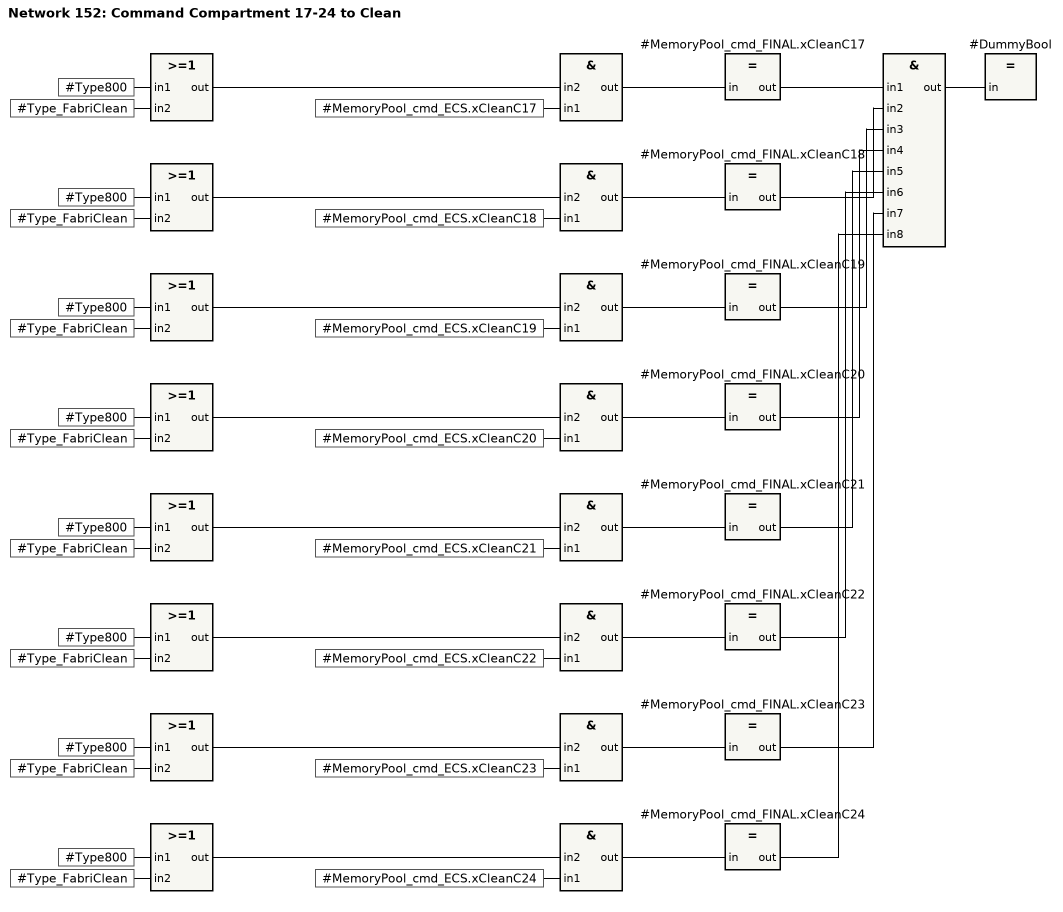
   #MemoryPool_cmd_FINAL.xCleanC17 := (#Type800 OR #Type_FabriClean) AND #MemoryPool_cmd_ECS.xCleanC17;
   #MemoryPool_cmd_FINAL.xCleanC18 := (#Type800 OR #Type_FabriClean) AND #MemoryPool_cmd_ECS.xCleanC18;
   #MemoryPool_cmd_FINAL.xCleanC19 := (#Type800 OR #Type_FabriClean) AND #MemoryPool_cmd_ECS.xCleanC19;
   #MemoryPool_cmd_FINAL.xCleanC20 := (#Type800 OR #Type_FabriClean) AND #MemoryPool_cmd_ECS.xCleanC20;
   #MemoryPool_cmd_FINAL.xCleanC21 := (#Type800 OR #Type_FabriClean) AND #MemoryPool_cmd_ECS.xCleanC21;
   #MemoryPool_cmd_FINAL.xCleanC22 := (#Type800 OR #Type_FabriClean) AND #MemoryPool_cmd_ECS.xCleanC22;
   #MemoryPool_cmd_FINAL.xCleanC23 := (#Type800 OR #Type_FabriClean) AND #MemoryPool_cmd_ECS.xCleanC23;
   #MemoryPool_cmd_FINAL.xCleanC24 := (#Type800 OR #Type_FabriClean) AND #MemoryPool_cmd_ECS.xCleanC24;
   #DummyBool := #MemoryPool_cmd_FINAL.xCleanC17 AND #MemoryPool_cmd_FINAL.xCleanC18 AND #MemoryPool_cmd_FINAL.xCleanC19 AND #MemoryPool_cmd_FINAL.xCleanC20 AND #MemoryPool_cmd_FINAL.xCleanC21 AND #MemoryPool_cmd_FINAL.xCleanC22 AND #MemoryPool_cmd_FINAL.xCleanC23 AND #MemoryPool_cmd_FINAL.xCleanC24;
END_REGION

REGION Network 153: Reset Clean Command 1-8
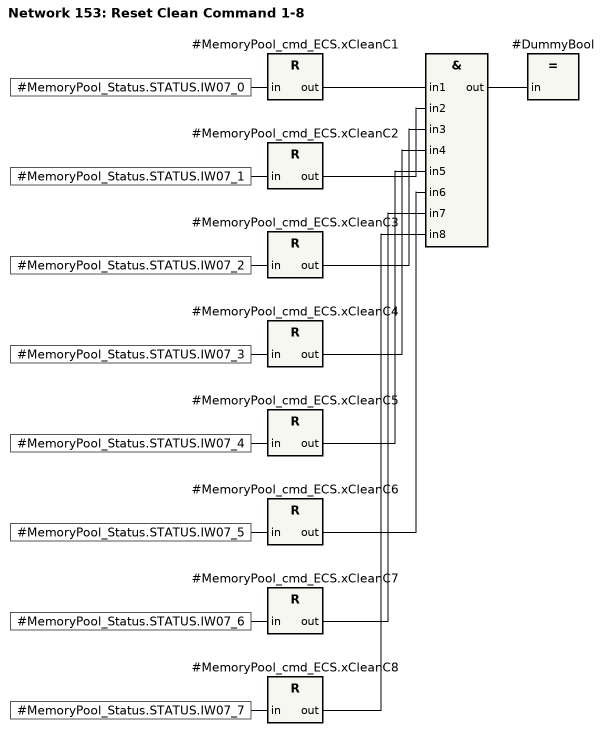
   IF #MemoryPool_Status.STATUS.IW07_0 THEN #MemoryPool_cmd_ECS.xCleanC1 := FALSE; END_IF;
   IF #MemoryPool_Status.STATUS.IW07_1 THEN #MemoryPool_cmd_ECS.xCleanC2 := FALSE; END_IF;
   IF #MemoryPool_Status.STATUS.IW07_2 THEN #MemoryPool_cmd_ECS.xCleanC3 := FALSE; END_IF;
   IF #MemoryPool_Status.STATUS.IW07_3 THEN #MemoryPool_cmd_ECS.xCleanC4 := FALSE; END_IF;
   IF #MemoryPool_Status.STATUS.IW07_4 THEN #MemoryPool_cmd_ECS.xCleanC5 := FALSE; END_IF;
   IF #MemoryPool_Status.STATUS.IW07_5 THEN #MemoryPool_cmd_ECS.xCleanC6 := FALSE; END_IF;
   IF #MemoryPool_Status.STATUS.IW07_6 THEN #MemoryPool_cmd_ECS.xCleanC7 := FALSE; END_IF;
   IF #MemoryPool_Status.STATUS.IW07_7 THEN #MemoryPool_cmd_ECS.xCleanC8 := FALSE; END_IF;
   #DummyBool := #MemoryPool_Status.STATUS.IW07_0 AND #MemoryPool_Status.STATUS.IW07_1 AND #MemoryPool_Status.STATUS.IW07_2 AND #MemoryPool_Status.STATUS.IW07_3 AND #MemoryPool_Status.STATUS.IW07_4 AND #MemoryPool_Status.STATUS.IW07_5 AND #MemoryPool_Status.STATUS.IW07_6 AND #MemoryPool_Status.STATUS.IW07_7;
END_REGION

REGION Network 154: Reset Clean Command 9-16
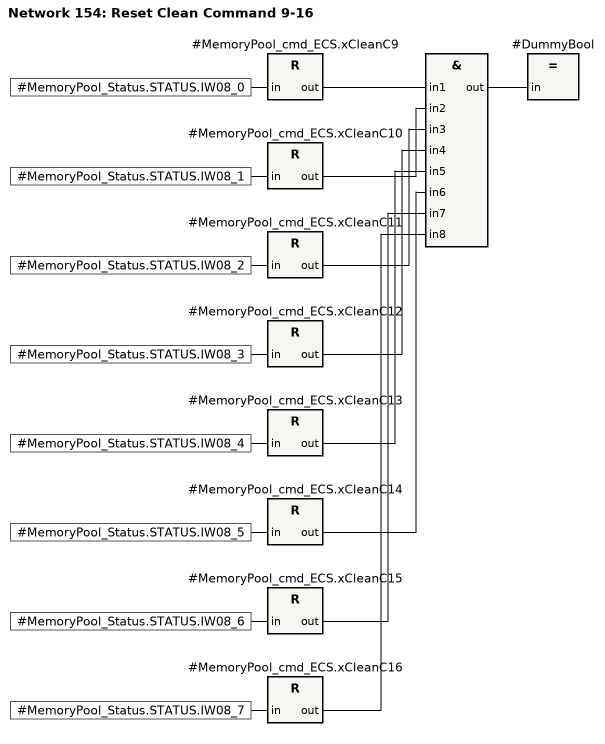
   IF #MemoryPool_Status.STATUS.IW08_0 THEN #MemoryPool_cmd_ECS.xCleanC9 := FALSE; END_IF;
   IF #MemoryPool_Status.STATUS.IW08_1 THEN #MemoryPool_cmd_ECS.xCleanC10 := FALSE; END_IF;
   IF #MemoryPool_Status.STATUS.IW08_2 THEN #MemoryPool_cmd_ECS.xCleanC11 := FALSE; END_IF;
   IF #MemoryPool_Status.STATUS.IW08_3 THEN #MemoryPool_cmd_ECS.xCleanC12 := FALSE; END_IF;
   IF #MemoryPool_Status.STATUS.IW08_4 THEN #MemoryPool_cmd_ECS.xCleanC13 := FALSE; END_IF;
   IF #MemoryPool_Status.STATUS.IW08_5 THEN #MemoryPool_cmd_ECS.xCleanC14 := FALSE; END_IF;
   IF #MemoryPool_Status.STATUS.IW08_6 THEN #MemoryPool_cmd_ECS.xCleanC15 := FALSE; END_IF;
   IF #MemoryPool_Status.STATUS.IW08_7 THEN #MemoryPool_cmd_ECS.xCleanC16 := FALSE; END_IF;
   #DummyBool := #MemoryPool_Status.STATUS.IW08_0 AND #MemoryPool_Status.STATUS.IW08_1 AND #MemoryPool_Status.STATUS.IW08_2 AND #MemoryPool_Status.STATUS.IW08_3 AND #MemoryPool_Status.STATUS.IW08_4 AND #MemoryPool_Status.STATUS.IW08_5 AND #MemoryPool_Status.STATUS.IW08_6 AND #MemoryPool_Status.STATUS.IW08_7;
END_REGION

REGION Network 155: Reset Clean Command 17-24
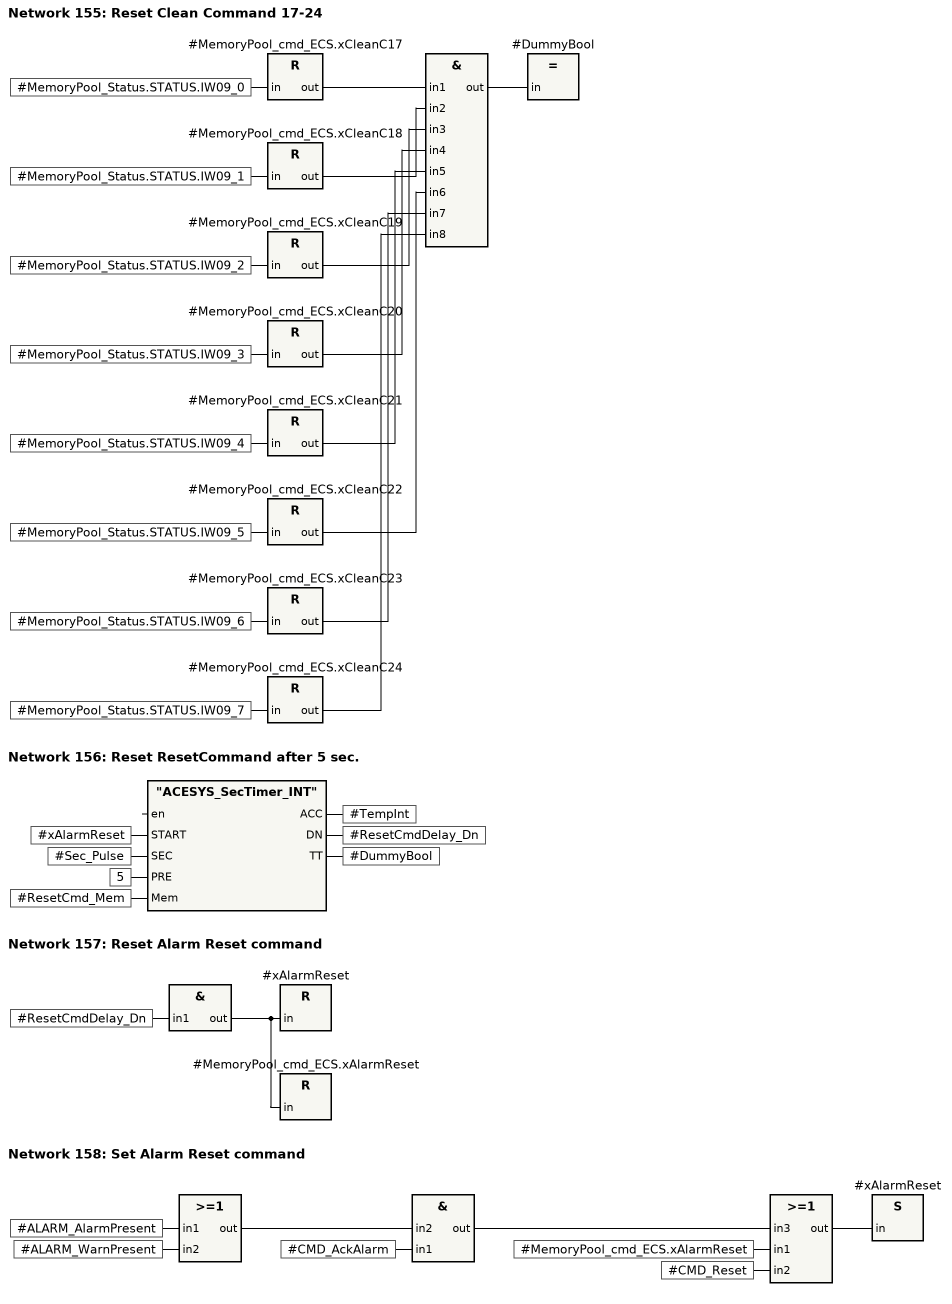
   IF #MemoryPool_Status.STATUS.IW09_0 THEN #MemoryPool_cmd_ECS.xCleanC17 := FALSE; END_IF;
   IF #MemoryPool_Status.STATUS.IW09_1 THEN #MemoryPool_cmd_ECS.xCleanC18 := FALSE; END_IF;
   IF #MemoryPool_Status.STATUS.IW09_2 THEN #MemoryPool_cmd_ECS.xCleanC19 := FALSE; END_IF;
   IF #MemoryPool_Status.STATUS.IW09_3 THEN #MemoryPool_cmd_ECS.xCleanC20 := FALSE; END_IF;
   IF #MemoryPool_Status.STATUS.IW09_4 THEN #MemoryPool_cmd_ECS.xCleanC21 := FALSE; END_IF;
   IF #MemoryPool_Status.STATUS.IW09_5 THEN #MemoryPool_cmd_ECS.xCleanC22 := FALSE; END_IF;
   IF #MemoryPool_Status.STATUS.IW09_6 THEN #MemoryPool_cmd_ECS.xCleanC23 := FALSE; END_IF;
   IF #MemoryPool_Status.STATUS.IW09_7 THEN #MemoryPool_cmd_ECS.xCleanC24 := FALSE; END_IF;
   #DummyBool := #MemoryPool_Status.STATUS.IW09_0 AND #MemoryPool_Status.STATUS.IW09_1 AND #MemoryPool_Status.STATUS.IW09_2 AND #MemoryPool_Status.STATUS.IW09_3 AND #MemoryPool_Status.STATUS.IW09_4 AND #MemoryPool_Status.STATUS.IW09_5 AND #MemoryPool_Status.STATUS.IW09_6 AND #MemoryPool_Status.STATUS.IW09_7;
END_REGION

REGION Network 156: Reset ResetCommand after 5 sec.
   "ACESYS_SecTimer_INT"(START := #xAlarmReset,
                         SEC := #Sec_Pulse,
                         PRE := 5,
                         Mem := #ResetCmd_Mem,
                         ACC => #TempInt,
                         DN => #ResetCmdDelay_Dn,
                         TT => #DummyBool);
END_REGION

REGION Network 157: Reset Alarm Reset command
   IF #ResetCmdDelay_Dn THEN
       #xAlarmReset := FALSE;
       #MemoryPool_cmd_ECS.xAlarmReset := FALSE;
   END_IF;
END_REGION

REGION Network 158: Set Alarm Reset command
   IF ((#ALARM_AlarmPresent OR #ALARM_WarnPresent) AND #CMD_AckAlarm) OR #MemoryPool_cmd_ECS.xAlarmReset OR #CMD_Reset THEN
       #xAlarmReset := TRUE;
   END_IF;
END_REGION

REGION Network 159
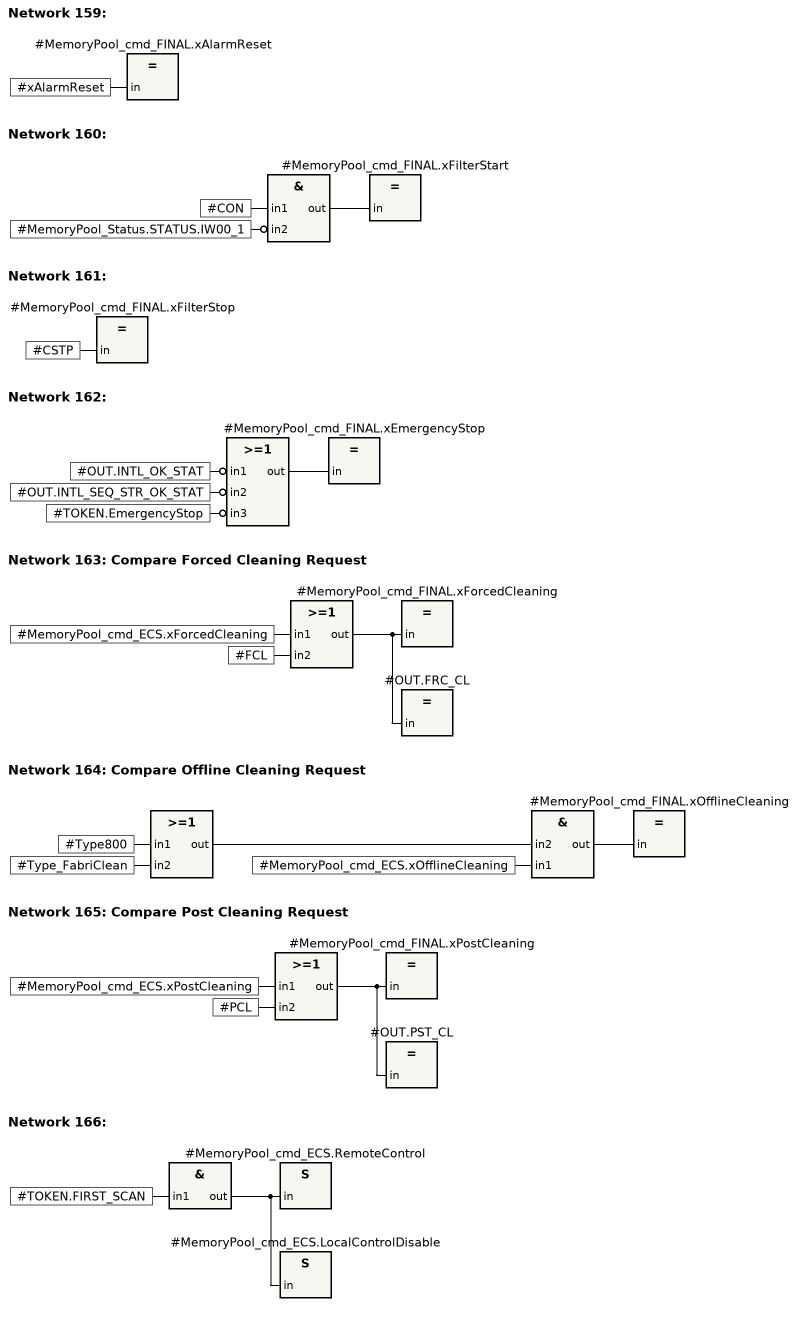
   #MemoryPool_cmd_FINAL.xAlarmReset := #xAlarmReset;
END_REGION

REGION Network 160
   #MemoryPool_cmd_FINAL.xFilterStart := #CON AND NOT #MemoryPool_Status.STATUS.IW00_1;
END_REGION

REGION Network 161
   #MemoryPool_cmd_FINAL.xFilterStop := #CSTP;
END_REGION

REGION Network 162
   #MemoryPool_cmd_FINAL.xEmergencyStop := NOT #OUT.INTL_OK_STAT OR NOT #OUT.INTL_SEQ_STR_OK_STAT OR NOT #TOKEN.EmergencyStop;
END_REGION

REGION Network 163: Compare Forced Cleaning Request
   #MemoryPool_cmd_FINAL.xForcedCleaning := #MemoryPool_cmd_ECS.xForcedCleaning OR #FCL;
   #OUT.FRC_CL := #MemoryPool_cmd_FINAL.xForcedCleaning;
END_REGION

REGION Network 164: Compare Offline Cleaning Request
   #MemoryPool_cmd_FINAL.xOfflineCleaning := (#Type800 OR #Type_FabriClean) AND #MemoryPool_cmd_ECS.xOfflineCleaning;
END_REGION

REGION Network 165: Compare Post Cleaning Request
   #MemoryPool_cmd_FINAL.xPostCleaning := #MemoryPool_cmd_ECS.xPostCleaning OR #PCL;
   #OUT.PST_CL := #MemoryPool_cmd_FINAL.xPostCleaning;
END_REGION

REGION Network 166
   IF #TOKEN.FIRST_SCAN THEN
       #MemoryPool_cmd_ECS.RemoteControl := TRUE;
       #MemoryPool_cmd_ECS.LocalControlDisable := TRUE;
   END_IF;
END_REGION

REGION Network 167
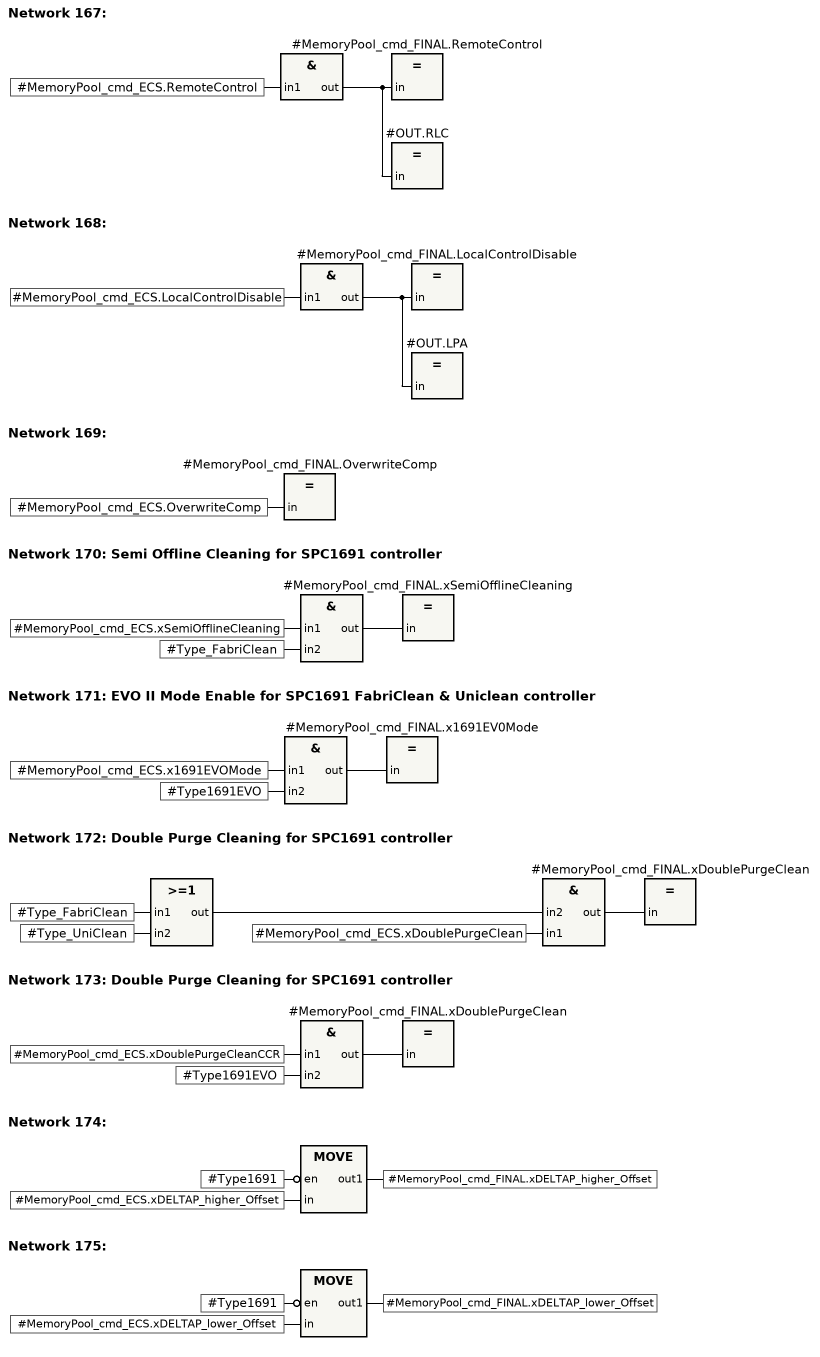
   #MemoryPool_cmd_FINAL.RemoteControl := #MemoryPool_cmd_ECS.RemoteControl;
   #OUT.RLC := #MemoryPool_cmd_ECS.RemoteControl;
END_REGION

REGION Network 168
   #MemoryPool_cmd_FINAL.LocalControlDisable := #MemoryPool_cmd_ECS.LocalControlDisable;
   #OUT.LPA := #MemoryPool_cmd_ECS.LocalControlDisable;
END_REGION

REGION Network 169
   #MemoryPool_cmd_FINAL.OverwriteComp := #MemoryPool_cmd_ECS.OverwriteComp;
END_REGION

REGION Network 170: Semi Offline Cleaning for SPC1691 controller
   #MemoryPool_cmd_FINAL.xSemiOfflineCleaning := #MemoryPool_cmd_ECS.xSemiOfflineCleaning AND #Type_FabriClean;
END_REGION

REGION Network 171: EVO II Mode Enable for SPC1691 FabriClean & Uniclean controller
   // Build 007 - 03.12.2020 (VIV-IN): EVO II Mode Enable for SPC1691 FabriClean & 
   // UniClean controller - Newly Added
   #MemoryPool_cmd_FINAL.x1691EV0Mode := #MemoryPool_cmd_ECS.x1691EVOMode AND #Type1691EVO;
END_REGION

REGION Network 172: Double Purge Cleaning for SPC1691 controller
   // Build 007 - 03.12.2020 (VIV-IN): Type UniClean also added
   #MemoryPool_cmd_FINAL.xDoublePurgeClean := (#Type_FabriClean OR #Type_UniClean) AND #MemoryPool_cmd_ECS.xDoublePurgeClean;
END_REGION

REGION Network 173: Double Purge Cleaning for SPC1691 controller
   // Build 007 - 03.12.2020 (VIV-IN): EVO Mode Double Purge Cleaning Continuous 
   // Cycle Request for SPC1691 FabriClean and UniClean controller - Newly Added
   #MemoryPool_cmd_FINAL.xDoublePurgeClean := #MemoryPool_cmd_ECS.xDoublePurgeCleanCCR AND #Type1691EVO;
END_REGION

REGION Network 174
   IF NOT #Type1691 THEN
       #MemoryPool_cmd_FINAL.xDELTAP_higher_Offset := #MemoryPool_cmd_ECS.xDELTAP_higher_Offset;
   END_IF;
END_REGION

REGION Network 175
   IF NOT #Type1691 THEN
       #MemoryPool_cmd_FINAL.xDELTAP_lower_Offset := #MemoryPool_cmd_ECS.xDELTAP_lower_Offset;
   END_IF;
END_REGION

REGION Network 176
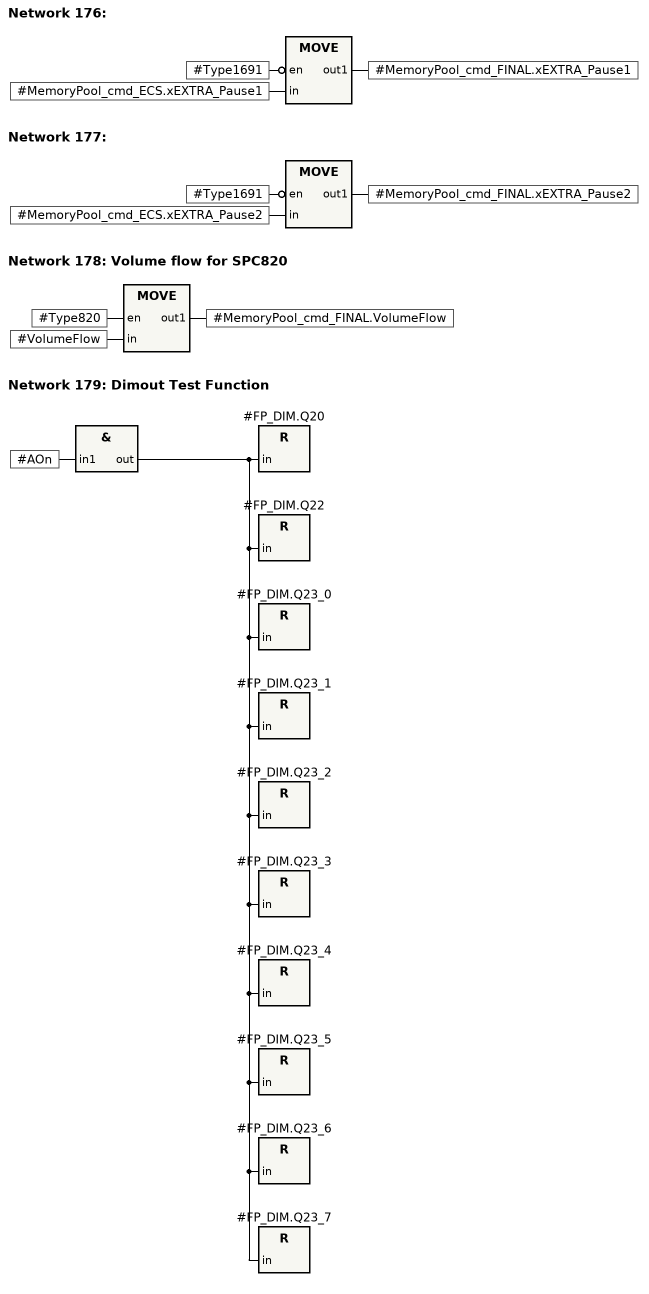
   IF NOT #Type1691 THEN #MemoryPool_cmd_FINAL.xEXTRA_Pause1 := #MemoryPool_cmd_ECS.xEXTRA_Pause1; END_IF;
END_REGION

REGION Network 177
   IF NOT #Type1691 THEN #MemoryPool_cmd_FINAL.xEXTRA_Pause2 := #MemoryPool_cmd_ECS.xEXTRA_Pause2; END_IF;
END_REGION

REGION Network 178: Volume flow for SPC820
   IF #Type820 THEN #MemoryPool_cmd_FINAL.VolumeFlow := #VolumeFlow; END_IF;
END_REGION

REGION Network 179: Dimout Test Function
   IF #AOn THEN
       #FP_DIM.Q20 := FALSE;
       #FP_DIM.Q22 := FALSE;
       #FP_DIM.Q23_0 := FALSE;
       #FP_DIM.Q23_1 := FALSE;
       #FP_DIM.Q23_2 := FALSE;
       #FP_DIM.Q23_3 := FALSE;
       #FP_DIM.Q23_4 := FALSE;
       #FP_DIM.Q23_5 := FALSE;
       #FP_DIM.Q23_6 := FALSE;
       #FP_DIM.Q23_7 := FALSE;
   END_IF;
END_REGION

REGION Network 180: Dimout test values/commands
   // Check for compartment number typed in
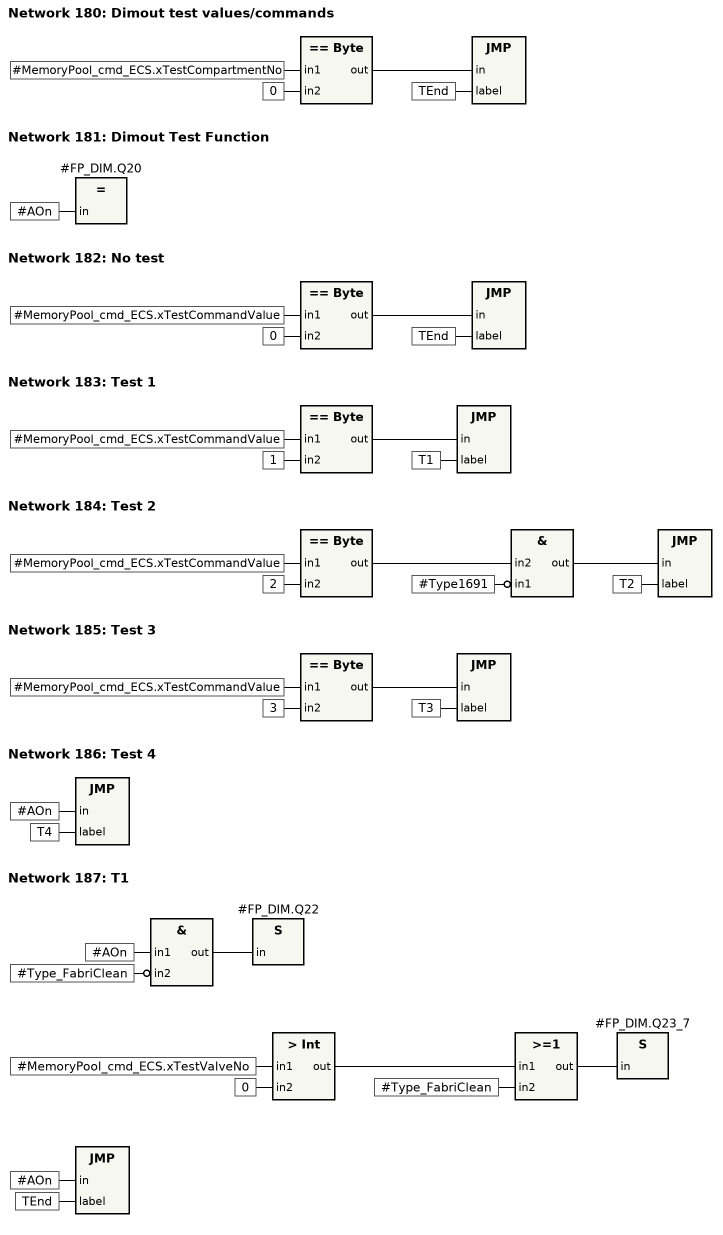
   IF #MemoryPool_cmd_ECS.xTestCompartmentNo = 0 THEN GOTO TEnd; END_IF;
END_REGION

REGION Network 181: Dimout Test Function
   #FP_DIM.Q20 := #AOn;
END_REGION

REGION Network 182: No test
   IF #MemoryPool_cmd_ECS.xTestCommandValue = 0 THEN GOTO TEnd; END_IF;
END_REGION

REGION Network 183: Test 1
   IF #MemoryPool_cmd_ECS.xTestCommandValue = 1 THEN GOTO T1; END_IF;
END_REGION

REGION Network 184: Test 2
   IF (#MemoryPool_cmd_ECS.xTestCommandValue = 2) AND NOT #Type1691 THEN GOTO T2; END_IF;
END_REGION

REGION Network 185: Test 3
   IF #MemoryPool_cmd_ECS.xTestCommandValue = 3 THEN GOTO T3; END_IF;
END_REGION

REGION Network 186: Test 4
   IF #AOn THEN GOTO T4; END_IF;
END_REGION

REGION Network 187: T1
   T1:
   IF #AOn AND NOT #Type_FabriClean THEN #FP_DIM.Q22 := TRUE; END_IF;
   IF (#MemoryPool_cmd_ECS.xTestValveNo > 0) OR #Type_FabriClean THEN #FP_DIM.Q23_7 := TRUE; END_IF;
   IF #AOn THEN GOTO TEnd; END_IF;
END_REGION

REGION Network 188: T2
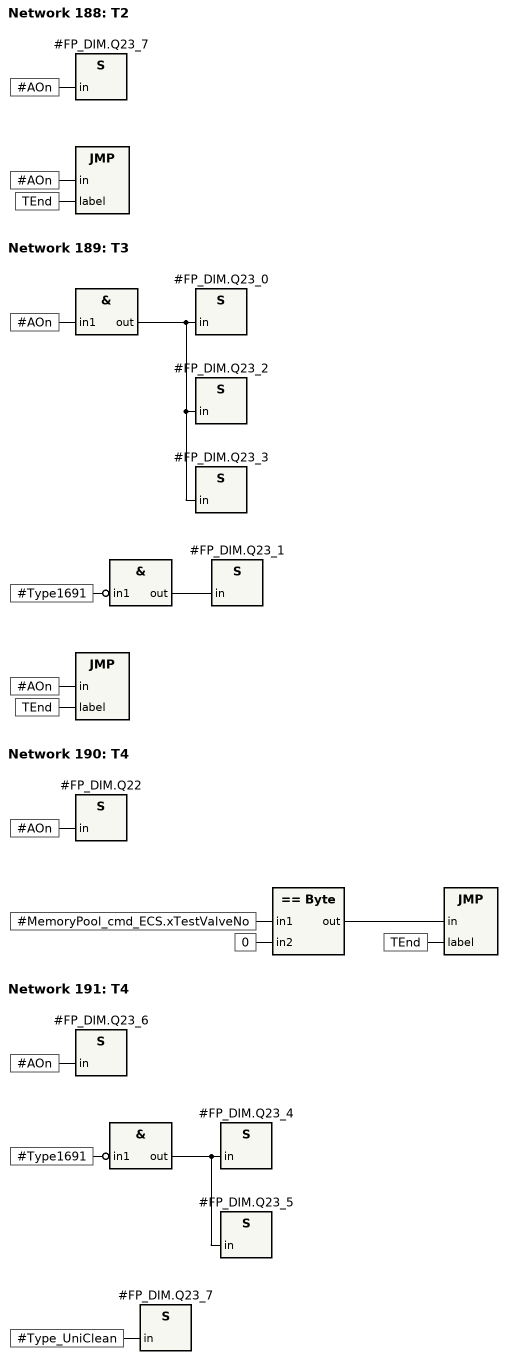
   T2:
   IF #AOn THEN
       #FP_DIM.Q23_7 := TRUE;
       GOTO TEnd;
   END_IF;
END_REGION

REGION Network 189: T3
   T3:
   IF #AOn THEN
       #FP_DIM.Q23_0 := TRUE;
       #FP_DIM.Q23_2 := TRUE;
       #FP_DIM.Q23_3 := TRUE;
   END_IF;
   IF NOT #Type1691 THEN #FP_DIM.Q23_1 := TRUE; END_IF;
   IF #AOn THEN GOTO TEnd; END_IF;
END_REGION

REGION Network 190: T4
   T4:
   IF #AOn THEN #FP_DIM.Q22 := TRUE; END_IF;
   IF #MemoryPool_cmd_ECS.xTestValveNo = 0 THEN GOTO TEnd; END_IF;
END_REGION

REGION Network 191: T4
   IF #AOn THEN #FP_DIM.Q23_6 := TRUE; END_IF;
   IF NOT #Type1691 THEN
       #FP_DIM.Q23_4 := TRUE;
       #FP_DIM.Q23_5 := TRUE;
   END_IF;
   IF #Type_UniClean THEN #FP_DIM.Q23_7 := TRUE; END_IF;
END_REGION

REGION Network 192
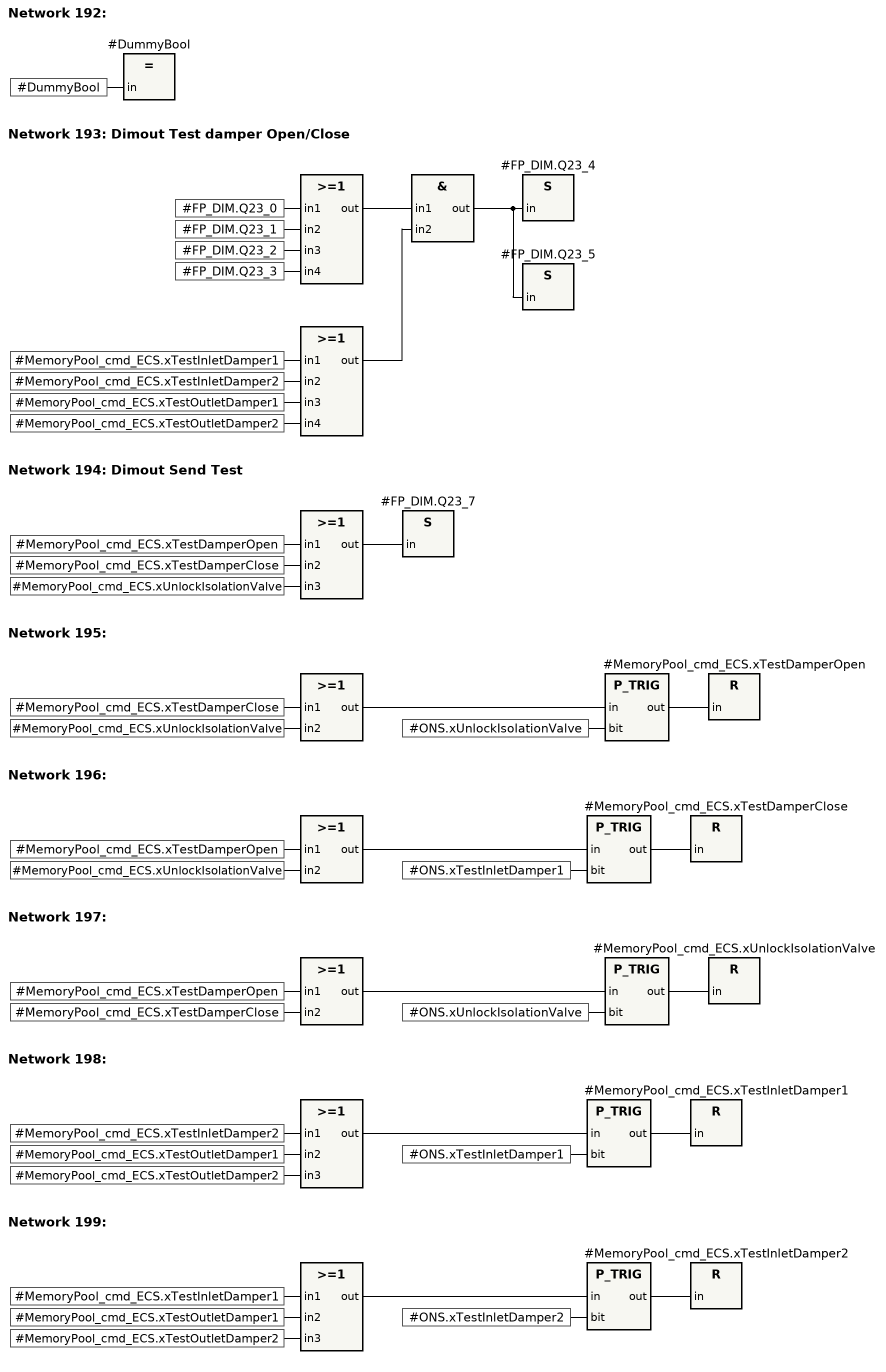
   TEnd:
   #DummyBool := #DummyBool;
END_REGION

REGION Network 193: Dimout Test damper Open/Close
   IF (#FP_DIM.Q23_0 OR #FP_DIM.Q23_1 OR #FP_DIM.Q23_2 OR #FP_DIM.Q23_3) AND (#MemoryPool_cmd_ECS.xTestInletDamper1 OR #MemoryPool_cmd_ECS.xTestInletDamper2 OR #MemoryPool_cmd_ECS.xTestOutletDamper1 OR #MemoryPool_cmd_ECS.xTestOutletDamper2) THEN
       #FP_DIM.Q23_4 := TRUE;
       #FP_DIM.Q23_5 := TRUE;
   END_IF;
END_REGION

REGION Network 194: Dimout Send Test
   IF #MemoryPool_cmd_ECS.xTestDamperOpen OR #MemoryPool_cmd_ECS.xTestDamperClose OR #MemoryPool_cmd_ECS.xUnlockIsolationValve THEN
       #FP_DIM.Q23_7 := TRUE;
   END_IF;
END_REGION

REGION Network 195
   #_w1 := #MemoryPool_cmd_ECS.xTestDamperClose OR #MemoryPool_cmd_ECS.xUnlockIsolationValve;
   #_w2 := #_w1 AND NOT #ONS.xUnlockIsolationValve;   // rising edge
   #ONS.xUnlockIsolationValve := #_w1;
   IF #_w2 THEN #MemoryPool_cmd_ECS.xTestDamperOpen := FALSE; END_IF;
END_REGION

REGION Network 196
   #_w1 := #MemoryPool_cmd_ECS.xTestDamperOpen OR #MemoryPool_cmd_ECS.xUnlockIsolationValve;
   #_w2 := #_w1 AND NOT #ONS.xTestInletDamper1;   // rising edge
   #ONS.xTestInletDamper1 := #_w1;
   IF #_w2 THEN #MemoryPool_cmd_ECS.xTestDamperClose := FALSE; END_IF;
END_REGION

REGION Network 197
   #_w1 := #MemoryPool_cmd_ECS.xTestDamperOpen OR #MemoryPool_cmd_ECS.xTestDamperClose;
   #_w2 := #_w1 AND NOT #ONS.xUnlockIsolationValve;   // rising edge
   #ONS.xUnlockIsolationValve := #_w1;
   IF #_w2 THEN #MemoryPool_cmd_ECS.xUnlockIsolationValve := FALSE; END_IF;
END_REGION

REGION Network 198
   #_w1 := #MemoryPool_cmd_ECS.xTestInletDamper2 OR #MemoryPool_cmd_ECS.xTestOutletDamper1 OR #MemoryPool_cmd_ECS.xTestOutletDamper2;
   #_w2 := #_w1 AND NOT #ONS.xTestInletDamper1;   // rising edge
   #ONS.xTestInletDamper1 := #_w1;
   IF #_w2 THEN #MemoryPool_cmd_ECS.xTestInletDamper1 := FALSE; END_IF;
END_REGION

REGION Network 199
   #_w1 := #MemoryPool_cmd_ECS.xTestInletDamper1 OR #MemoryPool_cmd_ECS.xTestOutletDamper1 OR #MemoryPool_cmd_ECS.xTestOutletDamper2;
   #_w2 := #_w1 AND NOT #ONS.xTestInletDamper2;   // rising edge
   #ONS.xTestInletDamper2 := #_w1;
   IF #_w2 THEN #MemoryPool_cmd_ECS.xTestInletDamper2 := FALSE; END_IF;
END_REGION

REGION Network 200
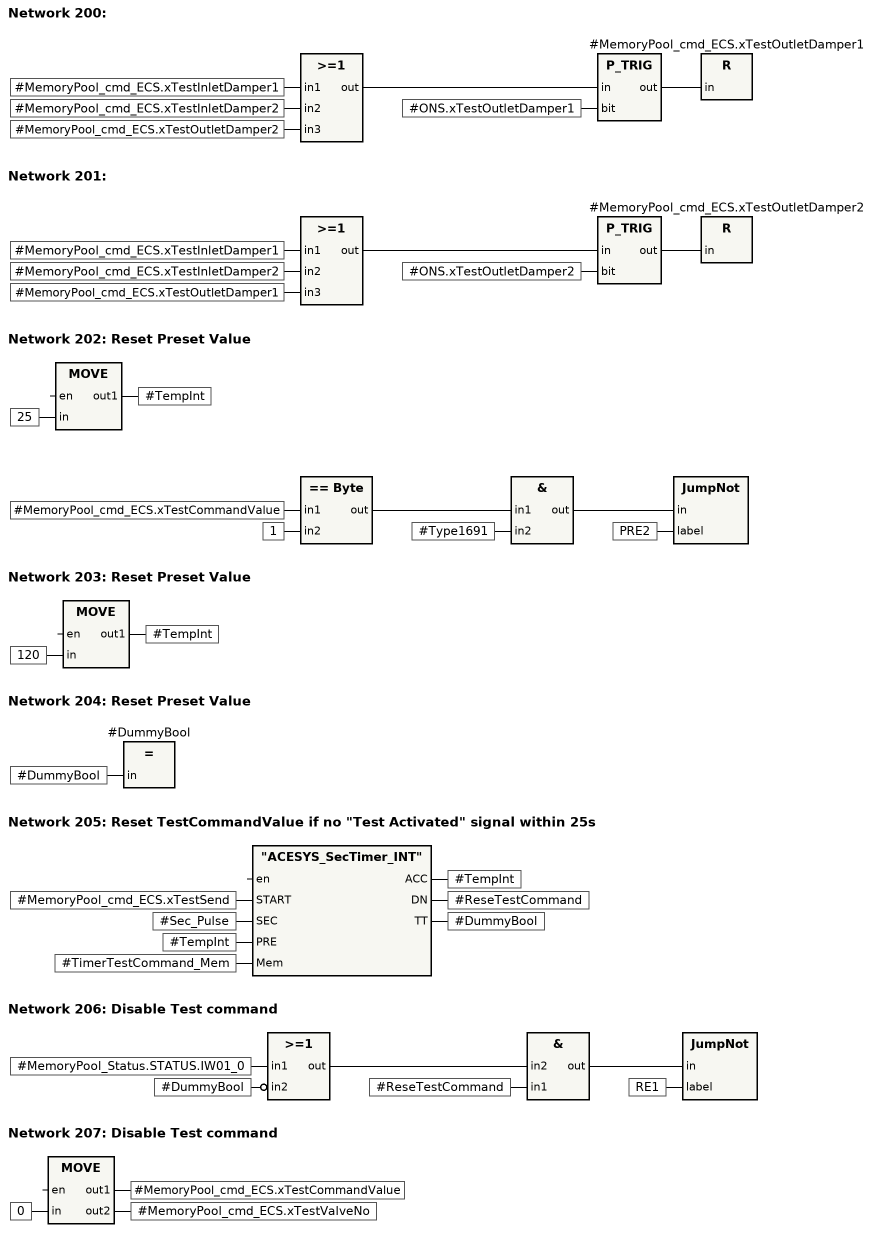
   #_w1 := #MemoryPool_cmd_ECS.xTestInletDamper1 OR #MemoryPool_cmd_ECS.xTestInletDamper2 OR #MemoryPool_cmd_ECS.xTestOutletDamper2;
   #_w2 := #_w1 AND NOT #ONS.xTestOutletDamper1;   // rising edge
   #ONS.xTestOutletDamper1 := #_w1;
   IF #_w2 THEN #MemoryPool_cmd_ECS.xTestOutletDamper1 := FALSE; END_IF;
END_REGION

REGION Network 201
   #_w1 := #MemoryPool_cmd_ECS.xTestInletDamper1 OR #MemoryPool_cmd_ECS.xTestInletDamper2 OR #MemoryPool_cmd_ECS.xTestOutletDamper1;
   #_w2 := #_w1 AND NOT #ONS.xTestOutletDamper2;   // rising edge
   #ONS.xTestOutletDamper2 := #_w1;
   IF #_w2 THEN #MemoryPool_cmd_ECS.xTestOutletDamper2 := FALSE; END_IF;
END_REGION

REGION Network 202: Reset Preset Value
   // - SPC1691 =>120s
   // - Hesch   =>25s
   // no SCL statement known for JumpNot: written as a call
   #TempInt := 25;
   JumpNot(in := (#MemoryPool_cmd_ECS.xTestCommandValue = 1) AND #Type1691, label := PRE2);
END_REGION

REGION Network 203: Reset Preset Value
   #TempInt := 120;
END_REGION

REGION Network 204: Reset Preset Value
   PRE2:
   #DummyBool := #DummyBool;
END_REGION

REGION Network 205: Reset TestCommandValue if no "Test Activated" signal within 25s
   "ACESYS_SecTimer_INT"(START := #MemoryPool_cmd_ECS.xTestSend,
                         SEC := #Sec_Pulse,
                         PRE := #TempInt,
                         Mem := #TimerTestCommand_Mem,
                         ACC => #TempInt,
                         DN => #ReseTestCommand,
                         TT => #DummyBool);
END_REGION

REGION Network 206: Disable Test command
   // Disable Test command once test activated is completed. This 
   // ensures that the command value is not always sent to the SPC
   // no SCL statement known for JumpNot: written as a call
   JumpNot(in := (#MemoryPool_Status.STATUS.IW01_0 OR NOT #DummyBool) AND #ReseTestCommand, label := RE1);
END_REGION

REGION Network 207: Disable Test command
   #MemoryPool_cmd_ECS.xTestCommandValue := 0;
   #MemoryPool_cmd_ECS.xTestValveNo := 0;
END_REGION

REGION Network 208: Disable Test command
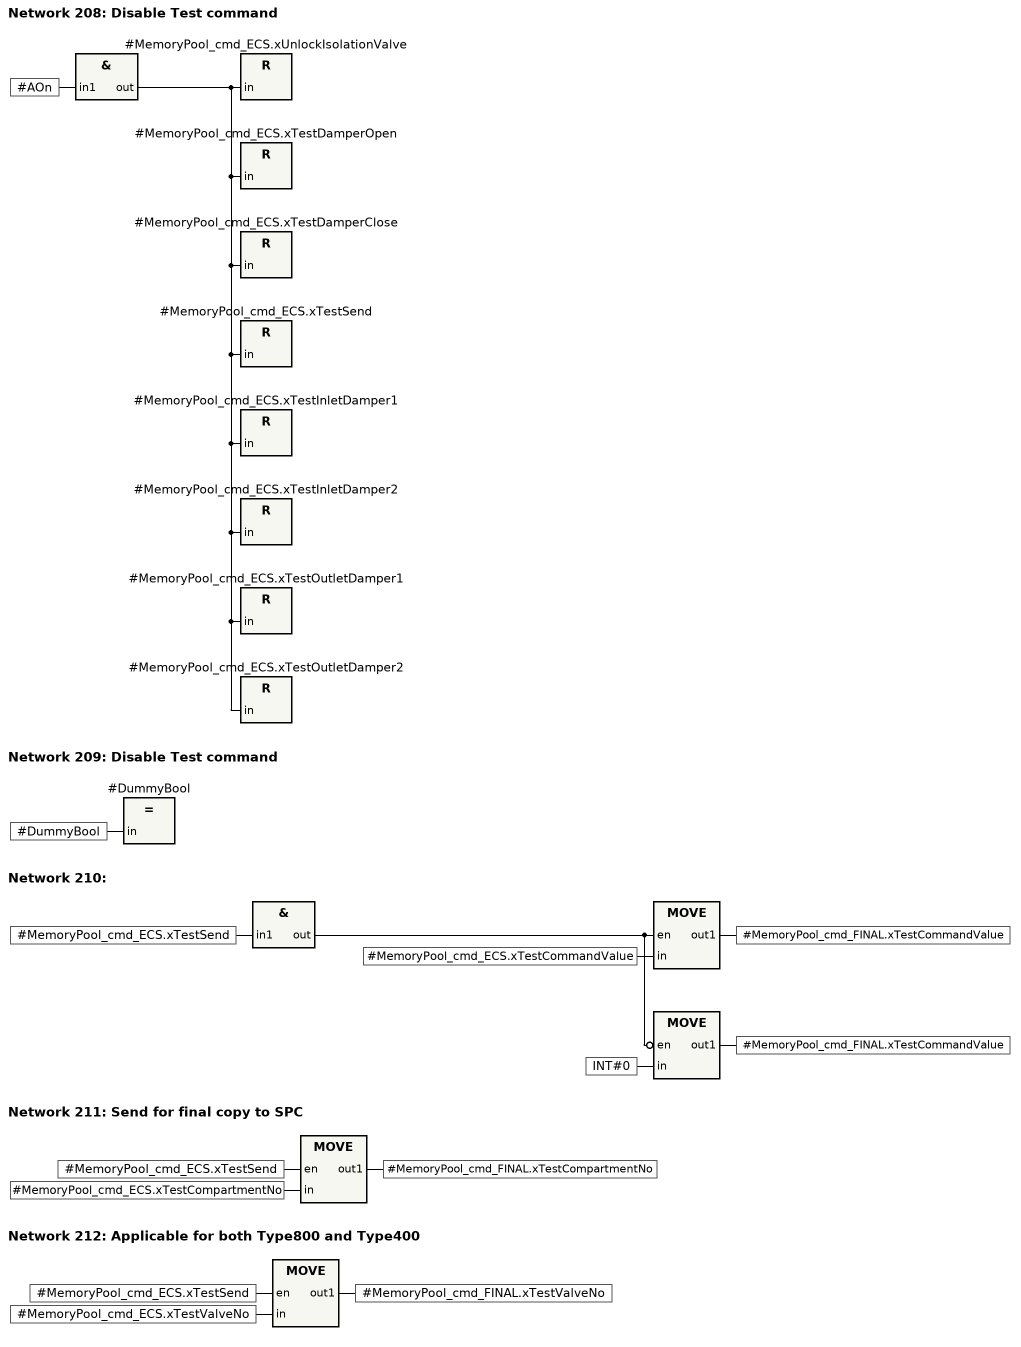
   IF #AOn THEN
       #MemoryPool_cmd_ECS.xUnlockIsolationValve := FALSE;
       #MemoryPool_cmd_ECS.xTestDamperOpen := FALSE;
       #MemoryPool_cmd_ECS.xTestDamperClose := FALSE;
       #MemoryPool_cmd_ECS.xTestSend := FALSE;
       #MemoryPool_cmd_ECS.xTestInletDamper1 := FALSE;
       #MemoryPool_cmd_ECS.xTestInletDamper2 := FALSE;
       #MemoryPool_cmd_ECS.xTestOutletDamper1 := FALSE;
       #MemoryPool_cmd_ECS.xTestOutletDamper2 := FALSE;
   END_IF;
END_REGION

REGION Network 209: Disable Test command
   RE1:
   #DummyBool := #DummyBool;
END_REGION

REGION Network 210
   IF #MemoryPool_cmd_ECS.xTestSend THEN
       #MemoryPool_cmd_FINAL.xTestCommandValue := #MemoryPool_cmd_ECS.xTestCommandValue;
   END_IF;
   IF NOT #MemoryPool_cmd_ECS.xTestSend THEN #MemoryPool_cmd_FINAL.xTestCommandValue := INT#0; END_IF;
END_REGION

REGION Network 211: Send for final copy to SPC
   // Applicable for Type 800 and 400. Type 400 is refered to as section
   IF #MemoryPool_cmd_ECS.xTestSend THEN
       #MemoryPool_cmd_FINAL.xTestCompartmentNo := #MemoryPool_cmd_ECS.xTestCompartmentNo;
   END_IF;
END_REGION

REGION Network 212: Applicable for both Type800 and Type400
   IF #MemoryPool_cmd_ECS.xTestSend THEN
       #MemoryPool_cmd_FINAL.xTestValveNo := #MemoryPool_cmd_ECS.xTestValveNo;
   END_IF;
END_REGION

REGION Network 213
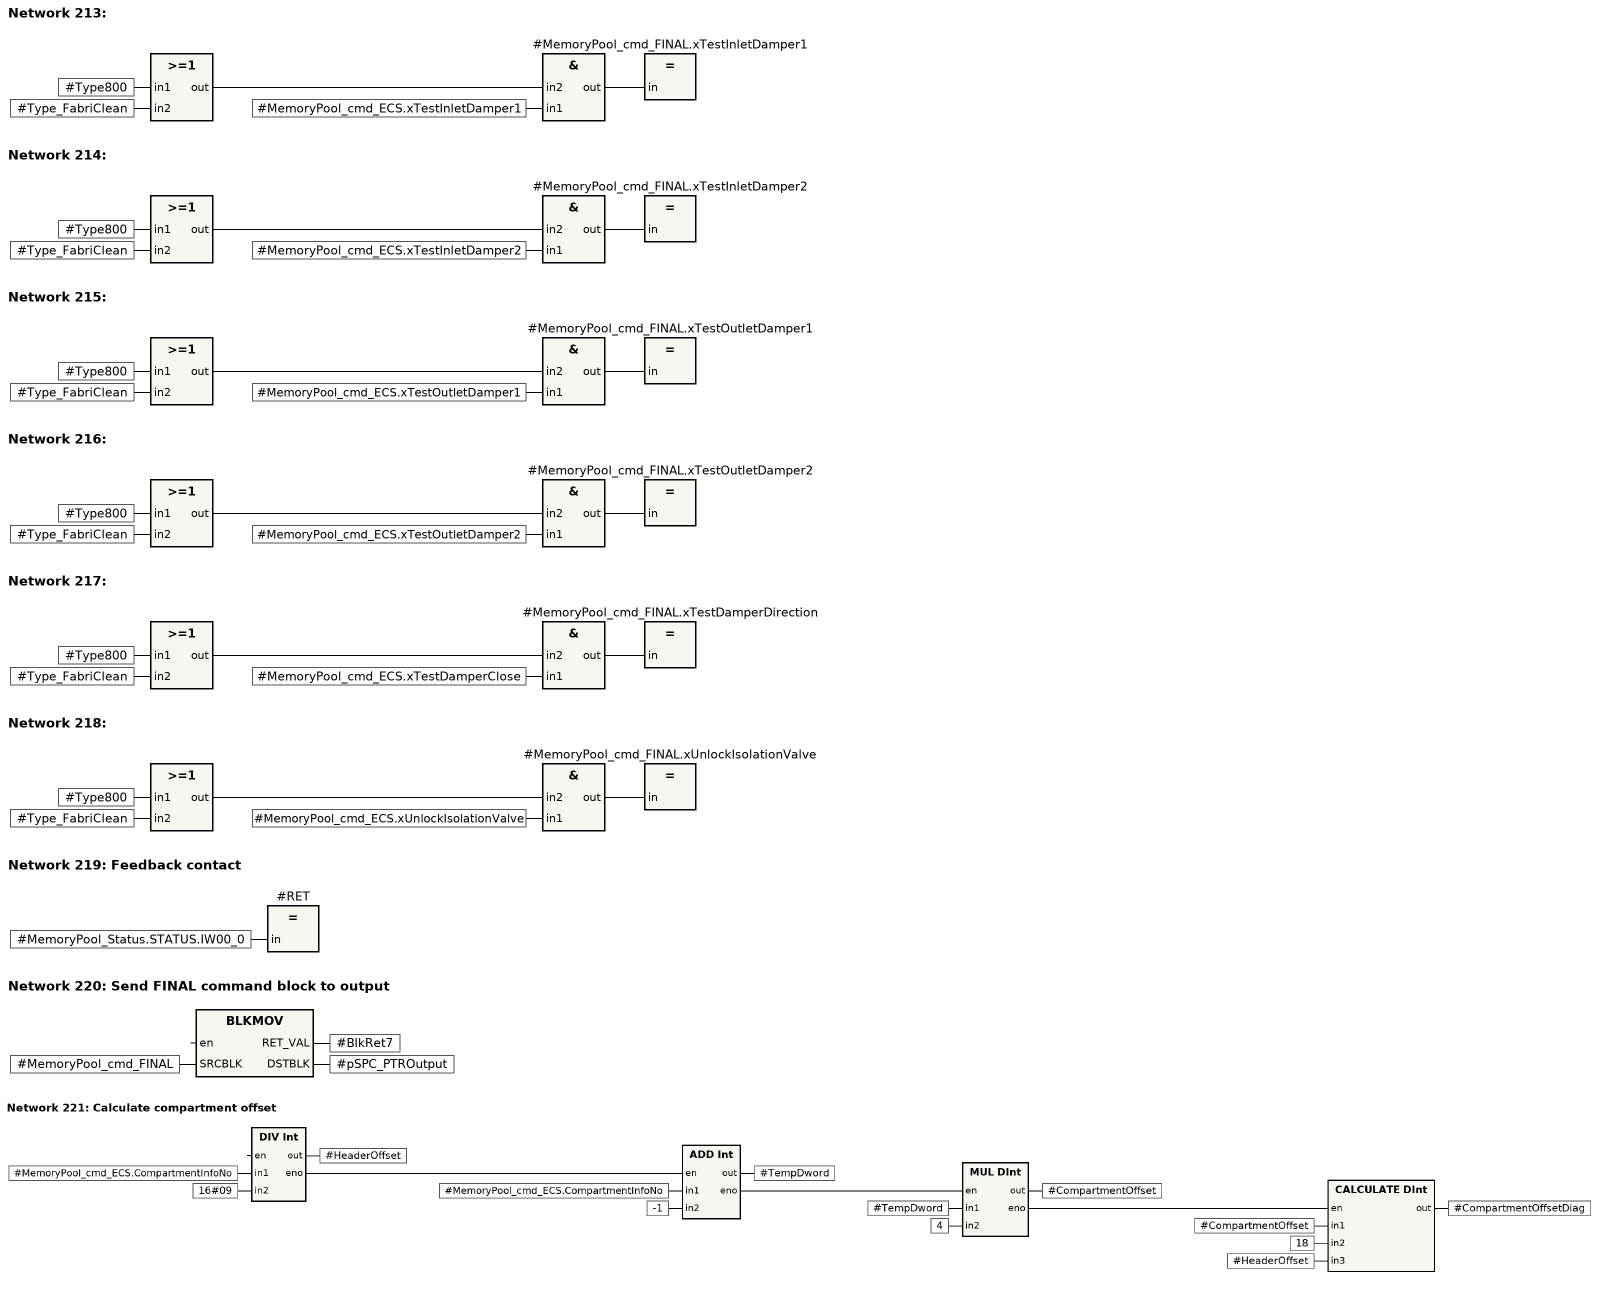
   #MemoryPool_cmd_FINAL.xTestInletDamper1 := (#Type800 OR #Type_FabriClean) AND #MemoryPool_cmd_ECS.xTestInletDamper1;
END_REGION

REGION Network 214
   #MemoryPool_cmd_FINAL.xTestInletDamper2 := (#Type800 OR #Type_FabriClean) AND #MemoryPool_cmd_ECS.xTestInletDamper2;
END_REGION

REGION Network 215
   #MemoryPool_cmd_FINAL.xTestOutletDamper1 := (#Type800 OR #Type_FabriClean) AND #MemoryPool_cmd_ECS.xTestOutletDamper1;
END_REGION

REGION Network 216
   #MemoryPool_cmd_FINAL.xTestOutletDamper2 := (#Type800 OR #Type_FabriClean) AND #MemoryPool_cmd_ECS.xTestOutletDamper2;
END_REGION

REGION Network 217
   #MemoryPool_cmd_FINAL.xTestDamperDirection := (#Type800 OR #Type_FabriClean) AND #MemoryPool_cmd_ECS.xTestDamperClose;
END_REGION

REGION Network 218
   #MemoryPool_cmd_FINAL.xUnlockIsolationValve := (#Type800 OR #Type_FabriClean) AND #MemoryPool_cmd_ECS.xUnlockIsolationValve;
END_REGION

REGION Network 219: Feedback contact
   #RET := #MemoryPool_Status.STATUS.IW00_0;
END_REGION

REGION Network 220: Send FINAL command block to output
   // Send FINAL command block to output. Destination length 30 BYTES.
   // byte 30..31 are not copied.
   #BlkRet7 := BLKMOV(SRCBLK := #MemoryPool_cmd_FINAL, DSTBLK => #pSPC_PTROutput);
END_REGION

REGION Network 221: Calculate compartment offset
   #HeaderOffset := #MemoryPool_cmd_ECS.CompartmentInfoNo / 16#09;
   #TempDword := #MemoryPool_cmd_ECS.CompartmentInfoNo + (-1);
   #CompartmentOffset := #TempDword * 4;
   #CompartmentOffsetDiag := #CompartmentOffset+18+#HeaderOffset;
END_REGION

REGION Network 222 (STL): Make pointer for compartment view Data
         LAR1;  //Make AR1 as Local Stack pointer

         L     16#10;  //Syntax ID
         T     B[AR1, P#0.0];

         L     16#02;  // Data Type= bytes
         T     B[AR1, P#1.0];

         L     4;
         T     W[AR1, P#2.0];  //BYTES TO TRANSFER

         L     #BlockInfo.DB_Number;
         T     W[AR1, P#4.0];  //Not Used

         L;  //Source offset (Variable for Node's)
         L     #CompartmentOffset;
         SLD   3;
         +D;
         L     16#8500_0000;
         -D;
         L     16#8400_0000;
         +D;
         T     D[AR1, P#6.0];  //..Store byte 6/7/8/9
END_REGION

REGION Network 223: Contruct data for ECS:COMPARTMENT_VIEW
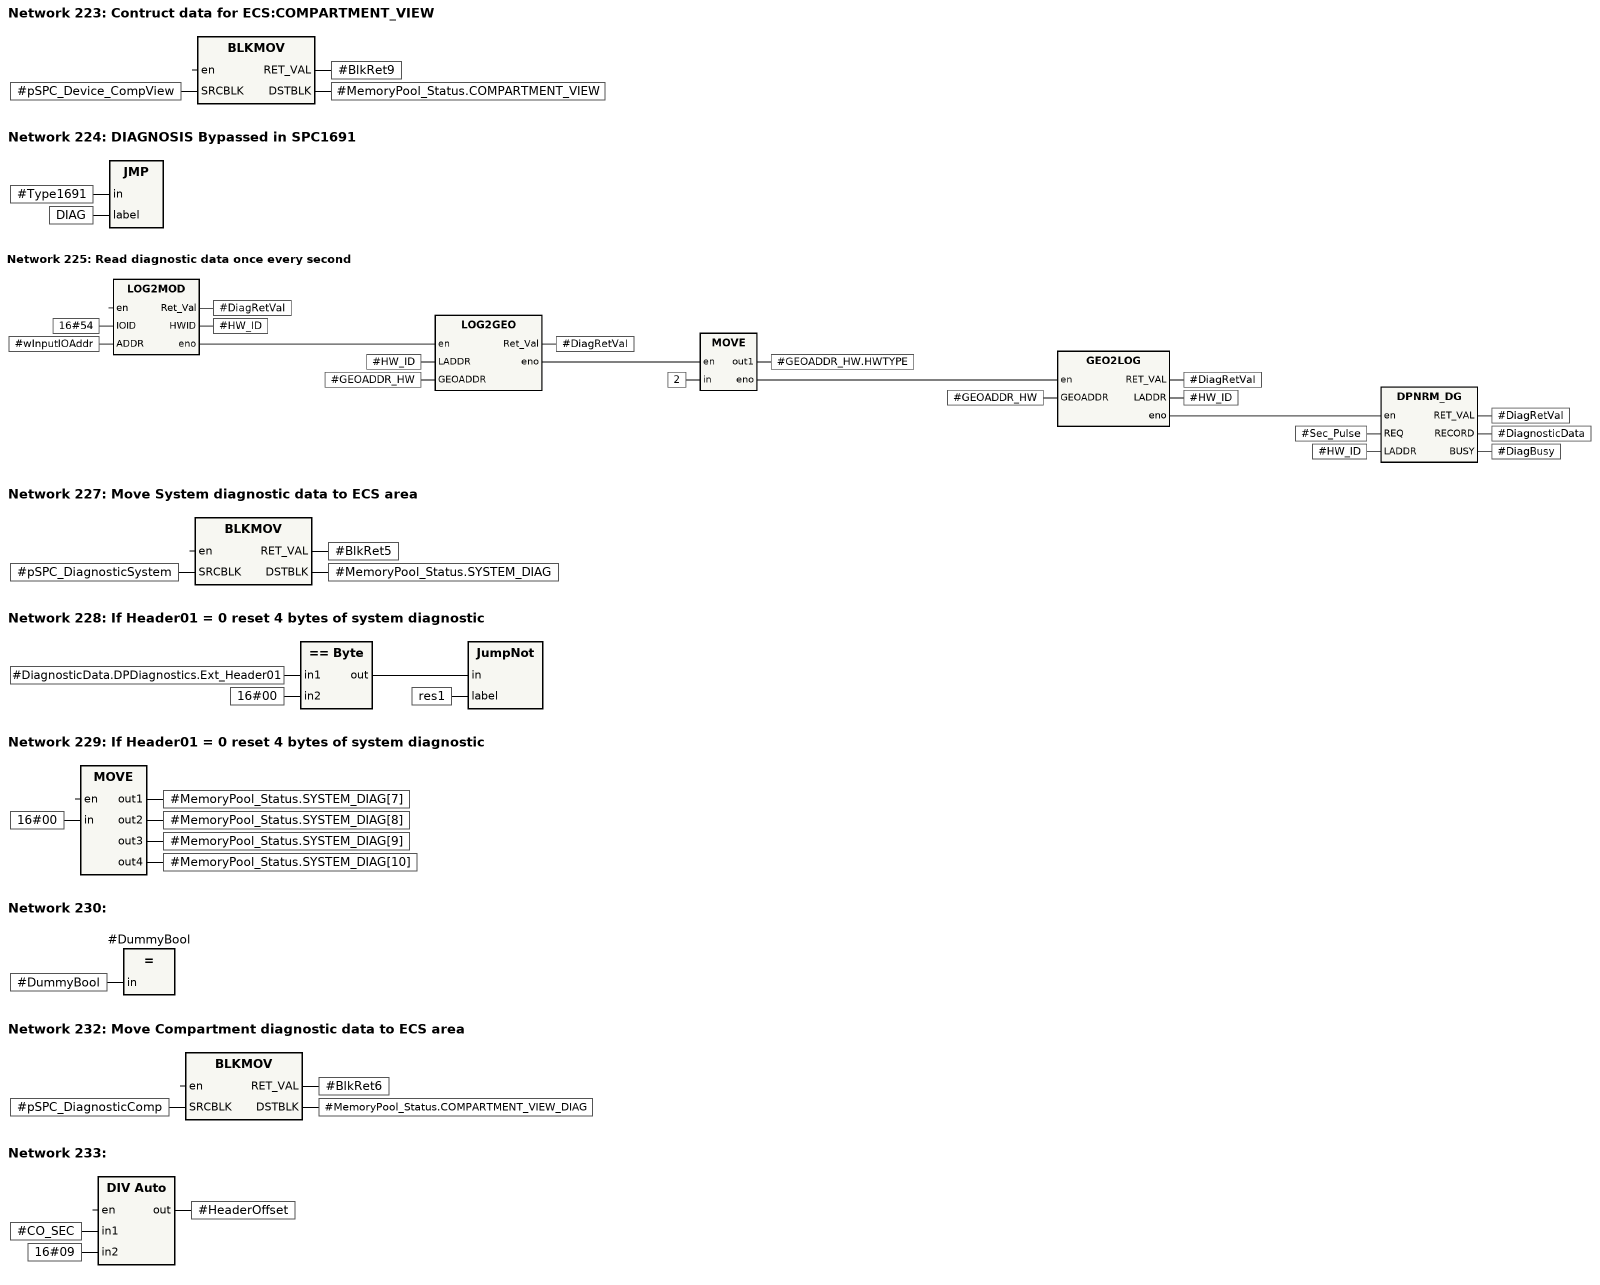
   #BlkRet9 := BLKMOV(SRCBLK := #pSPC_Device_CompView, DSTBLK => #MemoryPool_Status.COMPARTMENT_VIEW);
END_REGION

REGION Network 224: DIAGNOSIS Bypassed in SPC1691
   IF #Type1691 THEN GOTO DIAG; END_IF;
END_REGION

REGION Network 225: Read diagnostic data once every second
   // Build 004 - 08.May.2020 (MIA-US): Additional logic needed to retrieve HW_ID
   // ENO of a box is taken as its EN; it also drops when the box reports an error
   #DiagRetVal := LOG2MOD(IOID := 16#54, ADDR := #wInputIOAddr, HWID => #HW_ID);
   #DiagRetVal := LOG2GEO(LADDR := #HW_ID, GEOADDR := #GEOADDR_HW);
   #GEOADDR_HW.HWTYPE := 2;
   #DiagRetVal := GEO2LOG(GEOADDR := #GEOADDR_HW, LADDR => #HW_ID);
   #DiagRetVal := DPNRM_DG(REQ := #Sec_Pulse, LADDR := #HW_ID, RECORD => #DiagnosticData, BUSY => #DiagBusy);
END_REGION

REGION Network 226 (STL): POINTER CONSTRUCTION
   // Pointer for System Diagnostic Data
         LAR1;

         L     16#10;  //Syntax ID
         T     B[AR1, P#0.0];

         L     16#02;  // Data Type= bytes
         T     B[AR1, P#1.0];

         L     12;
         T     W[AR1, P#2.0];  //BYTES TO TRANSFER

         L     #BlockInfo.DB_Number;
         T     W[AR1, P#4.0];  //Not Used

         L;  // Source offset (Variable for Node's)
         L     16#8500_0000;
         -D;
         L     16#8400_0000;
         +D;
         T     D[AR1, P#6.0];  // ..Store byte 6/7/8/9
END_REGION

REGION Network 227: Move System diagnostic data to ECS area
   #BlkRet5 := BLKMOV(SRCBLK := #pSPC_DiagnosticSystem, DSTBLK => #MemoryPool_Status.SYSTEM_DIAG);
END_REGION

REGION Network 228: If Header01 = 0 reset 4 bytes of system diagnostic
   // no SCL statement known for JumpNot: written as a call
   JumpNot(in := #DiagnosticData.DPDiagnostics.Ext_Header01 = 16#00, label := res1);
END_REGION

REGION Network 229: If Header01 = 0 reset 4 bytes of system diagnostic
   #MemoryPool_Status.SYSTEM_DIAG[7] := 16#00;
   #MemoryPool_Status.SYSTEM_DIAG[8] := 16#00;
   #MemoryPool_Status.SYSTEM_DIAG[9] := 16#00;
   #MemoryPool_Status.SYSTEM_DIAG[10] := 16#00;
END_REGION

REGION Network 230
   res1:
   #DummyBool := #DummyBool;
END_REGION

REGION Network 231 (STL): Make pointer for Compartment Diagnostic Data
         LAR1;  //Make AR1 as Local Stack pointer

         L     16#10;  //Syntax ID
         T     B[AR1, P#0.0];

         L     16#02;  // Data Type= bytes
         T     B[AR1, P#1.0];

         L     4;
         T     W[AR1, P#2.0];  //BYTES TO TRANSFER

         L     #BlockInfo.DB_Number;
         T     W[AR1, P#4.0];  //Not Used

         L;  //Source offset (Variable for Node's)
         L     #CompartmentOffsetDiag;
         SLD   3;
         +D;
         L     16#8500_0000;
         -D;
         L     16#8400_0000;
         +D;
         T     D[AR1, P#6.0];  //..Store byte 6/7/8/9
END_REGION

REGION Network 232: Move Compartment diagnostic data to ECS area
   #BlkRet6 := BLKMOV(SRCBLK := #pSPC_DiagnosticComp, DSTBLK => #MemoryPool_Status.COMPARTMENT_VIEW_DIAG);
END_REGION

REGION Network 233
   #HeaderOffset := #CO_SEC / 16#09;
END_REGION

REGION Network 234: Calculation used in pointer for extra AI Diagnostic Data
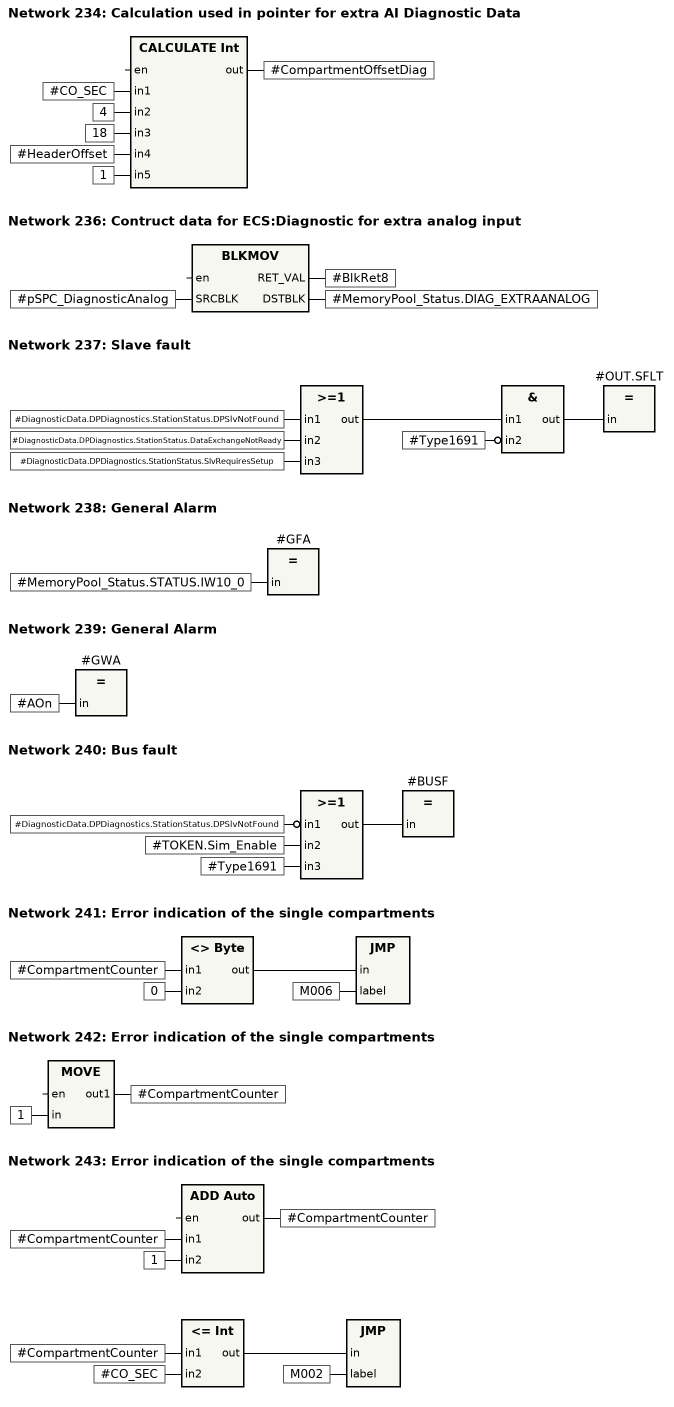
   #CompartmentOffsetDiag := (#CO_SEC*4)+18+#HeaderOffset+1;
END_REGION

REGION Network 235 (STL): Make pointer for extra AI Diagnostic Data
         LAR1;  //Make AR1 as Local Stack pointer

         L     16#10;  //Syntax ID
         T     B[AR1, P#0.0];

         L     16#02;  // Data Type= bytes
         T     B[AR1, P#1.0];

         L     2;
         T     W[AR1, P#2.0];  //BYTES TO TRANSFER

         L     #BlockInfo.DB_Number;
         T     W[AR1, P#4.0];  //Not Used

         L;  //Source offset (Variable for Node's)
         L     #CompartmentOffsetDiag;
         SLD   3;
         +D;
         L     16#8500_0000;
         -D;
         L     16#8400_0000;
         +D;
         T     D[AR1, P#6.0];  //..Store byte 6/7/8/9
END_REGION

REGION Network 236: Contruct data for ECS:Diagnostic for extra analog input
   #BlkRet8 := BLKMOV(SRCBLK := #pSPC_DiagnosticAnalog, DSTBLK => #MemoryPool_Status.DIAG_EXTRAANALOG);
END_REGION

REGION Network 237: Slave fault
   DIAG:
   #OUT.SFLT := (#DiagnosticData.DPDiagnostics.StationStatus.DPSlvNotFound OR #DiagnosticData.DPDiagnostics.StationStatus.DataExchangeNotReady OR #DiagnosticData.DPDiagnostics.StationStatus.SlvRequiresSetup) AND NOT #Type1691;
END_REGION

REGION Network 238: General Alarm
   #GFA := #MemoryPool_Status.STATUS.IW10_0;
END_REGION

REGION Network 239: General Alarm
   #GWA := #AOn;
END_REGION

REGION Network 240: Bus fault
   #BUSF := NOT #DiagnosticData.DPDiagnostics.StationStatus.DPSlvNotFound OR #TOKEN.Sim_Enable OR #Type1691;
END_REGION

REGION Network 241: Error indication of the single compartments
   IF #CompartmentCounter <> 0 THEN GOTO M006; END_IF;
END_REGION

REGION Network 242: Error indication of the single compartments
   #CompartmentCounter := 1;
END_REGION

REGION Network 243: Error indication of the single compartments
   // //Check one compartment each scan
   M006:
   #CompartmentCounter := #CompartmentCounter + 1;
   IF #CompartmentCounter <= #CO_SEC THEN GOTO M002; END_IF;
END_REGION

REGION Network 244: Error indication of the single compartments
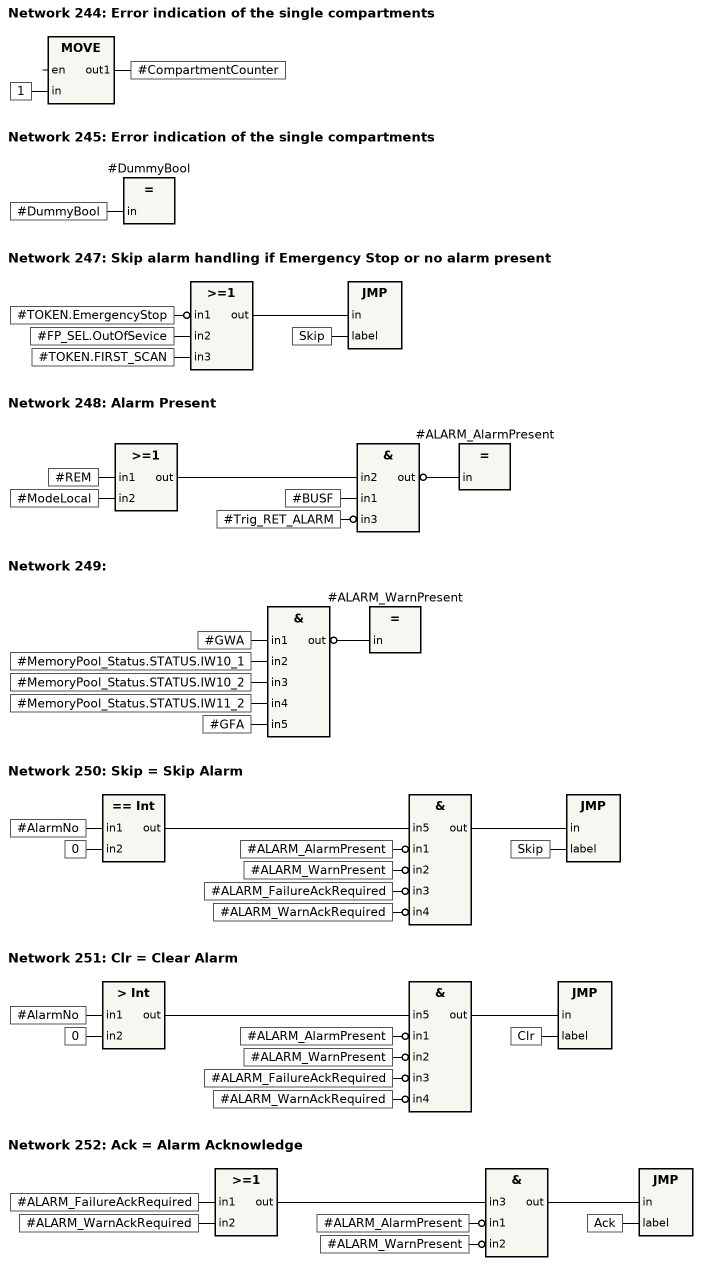
   #CompartmentCounter := 1;
END_REGION

REGION Network 245: Error indication of the single compartments
   M002:
   #DummyBool := #DummyBool;
END_REGION

REGION Network 246 (STL): Calculate pointer - Compartment Counter
         L     #CompartmentCounter;  //Calculate pointer
         L     1;
         -I;
         L     4;
         *I;
         +     3;
         SLD   3;
         L;  //Source offset
         +D;
         LAR1;
         L     B[AR1, P#0.0];  //Actual compartment valve no. malfunction
         L     0;
         ==I;
         JC    M004;  //Jump if no valve error

         L     #CompartmentCounter;  //
         L     1;
         -I;
         L;  //Source offset
         +D;
         LAR1;
         A     #AOn;
         S     [AR1, P#0.0];  //Set error bit
         JU    M003;

   M004: L     #CompartmentCounter;  //If no error reset error bit
         L     1;
         -I;
         L;  //Source offset
         +D;
         LAR1;
         A     #AOn;
         R     [AR1, P#0.0];  //Reset error bit
   M003: NOP   1;
END_REGION

REGION Network 247: Skip alarm handling if Emergency Stop or no alarm present
   // Skip = Skip Alarm
   IF NOT #TOKEN.EmergencyStop OR #FP_SEL.OutOfSevice OR #TOKEN.FIRST_SCAN THEN GOTO Skip; END_IF;
END_REGION

REGION Network 248: Alarm Present
   #ALARM_AlarmPresent := NOT ((#REM OR #ModeLocal) AND #BUSF AND NOT #Trig_RET_ALARM);
END_REGION

REGION Network 249
   #ALARM_WarnPresent := NOT (#GWA AND #MemoryPool_Status.STATUS.IW10_1 AND #MemoryPool_Status.STATUS.IW10_2 AND #MemoryPool_Status.STATUS.IW11_2 AND #GFA);
END_REGION

REGION Network 250: Skip = Skip Alarm
   IF (#AlarmNo = 0) AND NOT #ALARM_AlarmPresent AND NOT #ALARM_WarnPresent AND NOT #ALARM_FailureAckRequired AND NOT #ALARM_WarnAckRequired THEN
       GOTO Skip;
   END_IF;
END_REGION

REGION Network 251: Clr = Clear Alarm
   IF (#AlarmNo > 0) AND NOT #ALARM_AlarmPresent AND NOT #ALARM_WarnPresent AND NOT #ALARM_FailureAckRequired AND NOT #ALARM_WarnAckRequired THEN
       GOTO Clr;
   END_IF;
END_REGION

REGION Network 252: Ack = Alarm Acknowledge
   IF (#ALARM_FailureAckRequired OR #ALARM_WarnAckRequired) AND NOT #ALARM_AlarmPresent AND NOT #ALARM_WarnPresent THEN
       GOTO Ack;
   END_IF;
END_REGION

REGION Network 253: Bus Fault
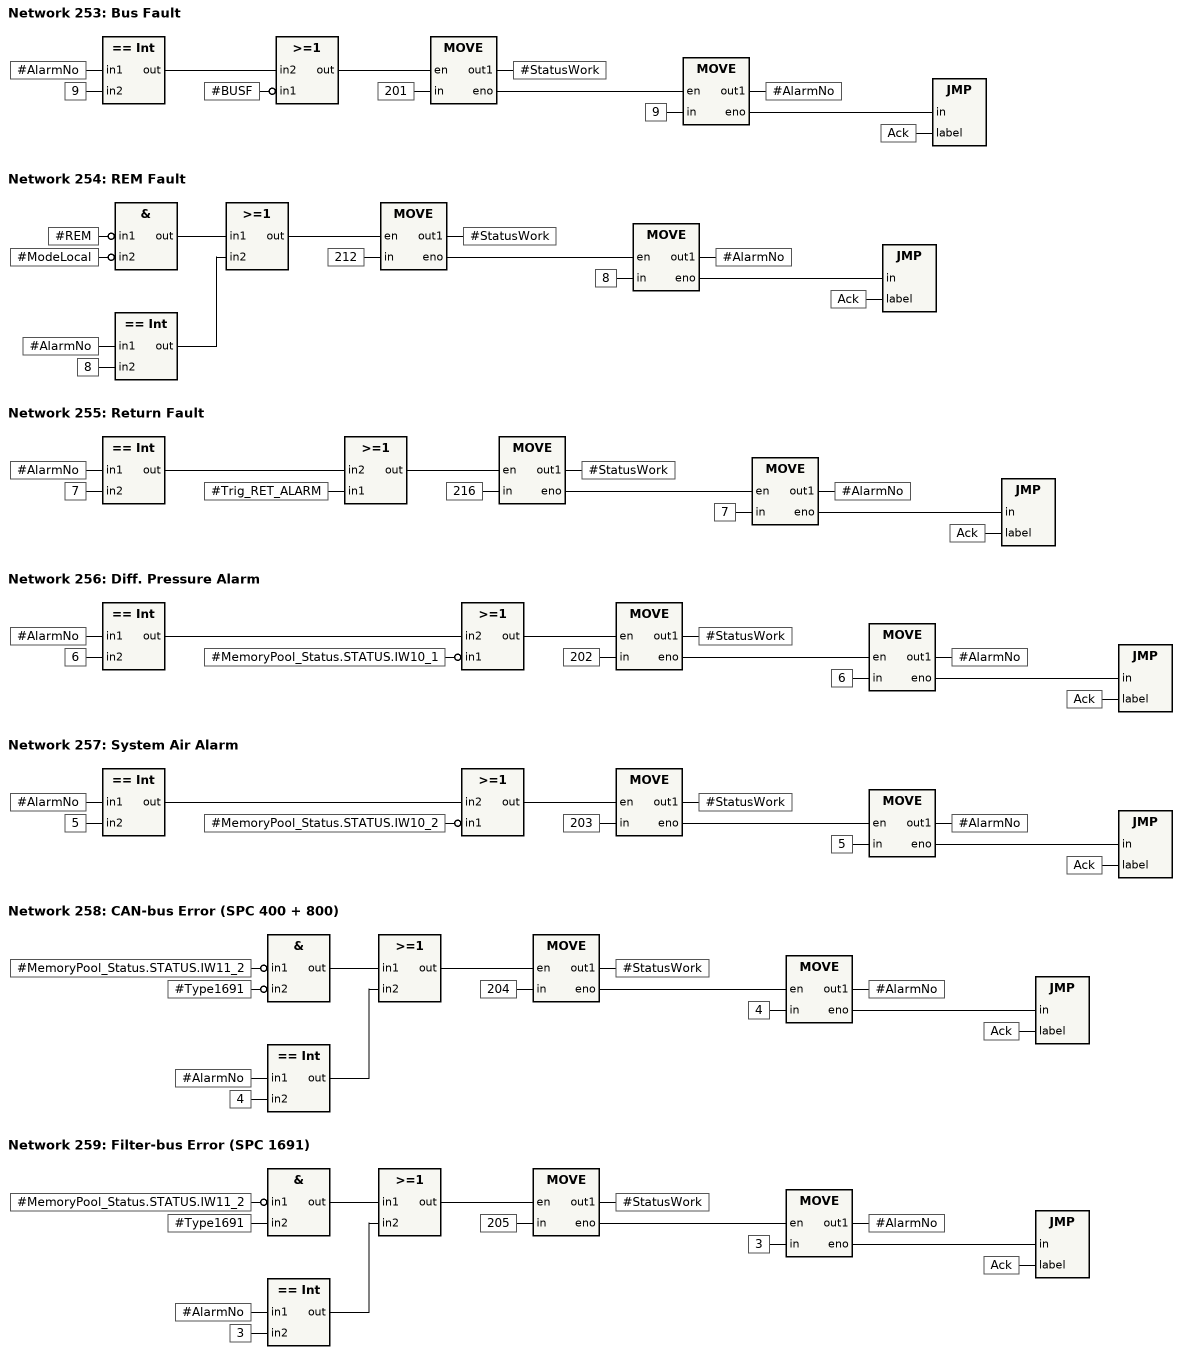
   // ENO of a box is taken as its EN; it also drops when the box reports an error
   #_w1 := (#AlarmNo = 9) OR NOT #BUSF;
   IF #_w1 THEN
       #StatusWork := 201;
       #AlarmNo := 9;
       GOTO Ack;
   END_IF;
END_REGION

REGION Network 254: REM Fault
   // ENO of a box is taken as its EN; it also drops when the box reports an error
   #_w1 := (NOT #REM AND NOT #ModeLocal) OR (#AlarmNo = 8);
   IF #_w1 THEN
       #StatusWork := 212;
       #AlarmNo := 8;
       GOTO Ack;
   END_IF;
END_REGION

REGION Network 255: Return Fault
   // ENO of a box is taken as its EN; it also drops when the box reports an error
   #_w1 := (#AlarmNo = 7) OR #Trig_RET_ALARM;
   IF #_w1 THEN
       #StatusWork := 216;
       #AlarmNo := 7;
       GOTO Ack;
   END_IF;
END_REGION

REGION Network 256: Diff. Pressure Alarm
   // ENO of a box is taken as its EN; it also drops when the box reports an error
   #_w1 := (#AlarmNo = 6) OR NOT #MemoryPool_Status.STATUS.IW10_1;
   IF #_w1 THEN
       #StatusWork := 202;
       #AlarmNo := 6;
       GOTO Ack;
   END_IF;
END_REGION

REGION Network 257: System Air Alarm
   // ENO of a box is taken as its EN; it also drops when the box reports an error
   #_w1 := (#AlarmNo = 5) OR NOT #MemoryPool_Status.STATUS.IW10_2;
   IF #_w1 THEN
       #StatusWork := 203;
       #AlarmNo := 5;
       GOTO Ack;
   END_IF;
END_REGION

REGION Network 258: CAN-bus Error (SPC 400 + 800)
   // ENO of a box is taken as its EN; it also drops when the box reports an error
   #_w1 := (NOT #MemoryPool_Status.STATUS.IW11_2 AND NOT #Type1691) OR (#AlarmNo = 4);
   IF #_w1 THEN
       #StatusWork := 204;
       #AlarmNo := 4;
       GOTO Ack;
   END_IF;
END_REGION

REGION Network 259: Filter-bus Error (SPC 1691)
   // ENO of a box is taken as its EN; it also drops when the box reports an error
   #_w1 := (NOT #MemoryPool_Status.STATUS.IW11_2 AND #Type1691) OR (#AlarmNo = 3);
   IF #_w1 THEN
       #StatusWork := 205;
       #AlarmNo := 3;
       GOTO Ack;
   END_IF;
END_REGION

REGION Network 260: GFA Fault
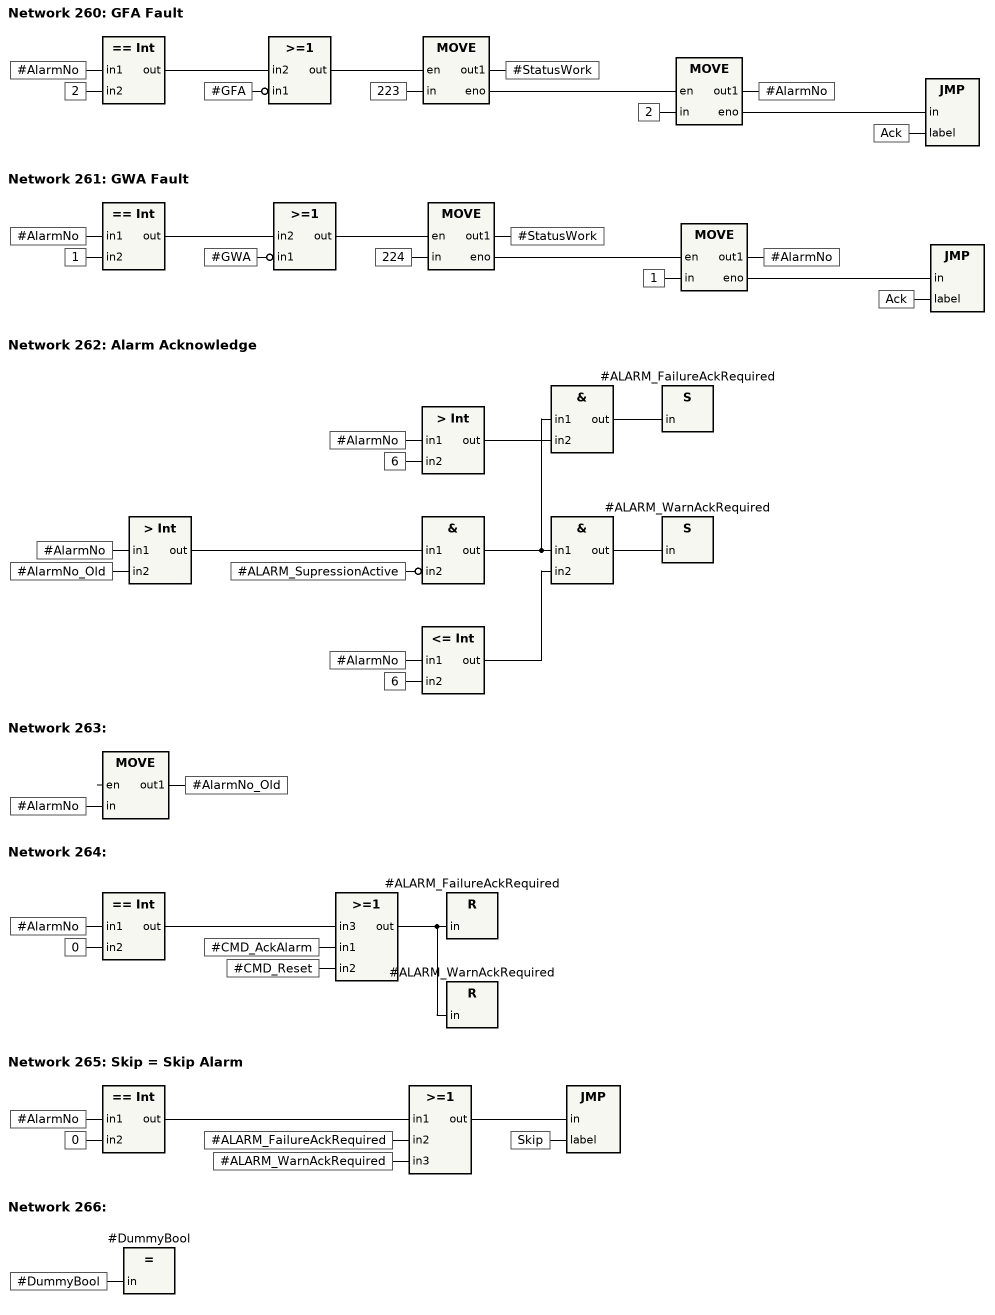
   // ENO of a box is taken as its EN; it also drops when the box reports an error
   #_w1 := (#AlarmNo = 2) OR NOT #GFA;
   IF #_w1 THEN
       #StatusWork := 223;
       #AlarmNo := 2;
       GOTO Ack;
   END_IF;
END_REGION

REGION Network 261: GWA Fault
   // ENO of a box is taken as its EN; it also drops when the box reports an error
   #_w1 := (#AlarmNo = 1) OR NOT #GWA;
   IF #_w1 THEN
       #StatusWork := 224;
       #AlarmNo := 1;
       GOTO Ack;
   END_IF;
END_REGION

REGION Network 262: Alarm Acknowledge
   // AlarmNo >6 Are made Warning
   Ack:
   #_w1 := (#AlarmNo > #AlarmNo_Old) AND NOT #ALARM_SupressionActive;
   IF #_w1 AND (#AlarmNo > 6) THEN #ALARM_FailureAckRequired := TRUE; END_IF;
   IF #_w1 AND (#AlarmNo <= 6) THEN #ALARM_WarnAckRequired := TRUE; END_IF;
END_REGION

REGION Network 263
   #AlarmNo_Old := #AlarmNo;
END_REGION

REGION Network 264
   IF (#AlarmNo = 0) OR #CMD_AckAlarm OR #CMD_Reset THEN
       #ALARM_FailureAckRequired := FALSE;
       #ALARM_WarnAckRequired := FALSE;
   END_IF;
END_REGION

REGION Network 265: Skip = Skip Alarm
   IF (#AlarmNo = 0) OR #ALARM_FailureAckRequired OR #ALARM_WarnAckRequired THEN GOTO Skip; END_IF;
END_REGION

REGION Network 266
   Clr:
   #DummyBool := #DummyBool;
END_REGION

REGION Network 267
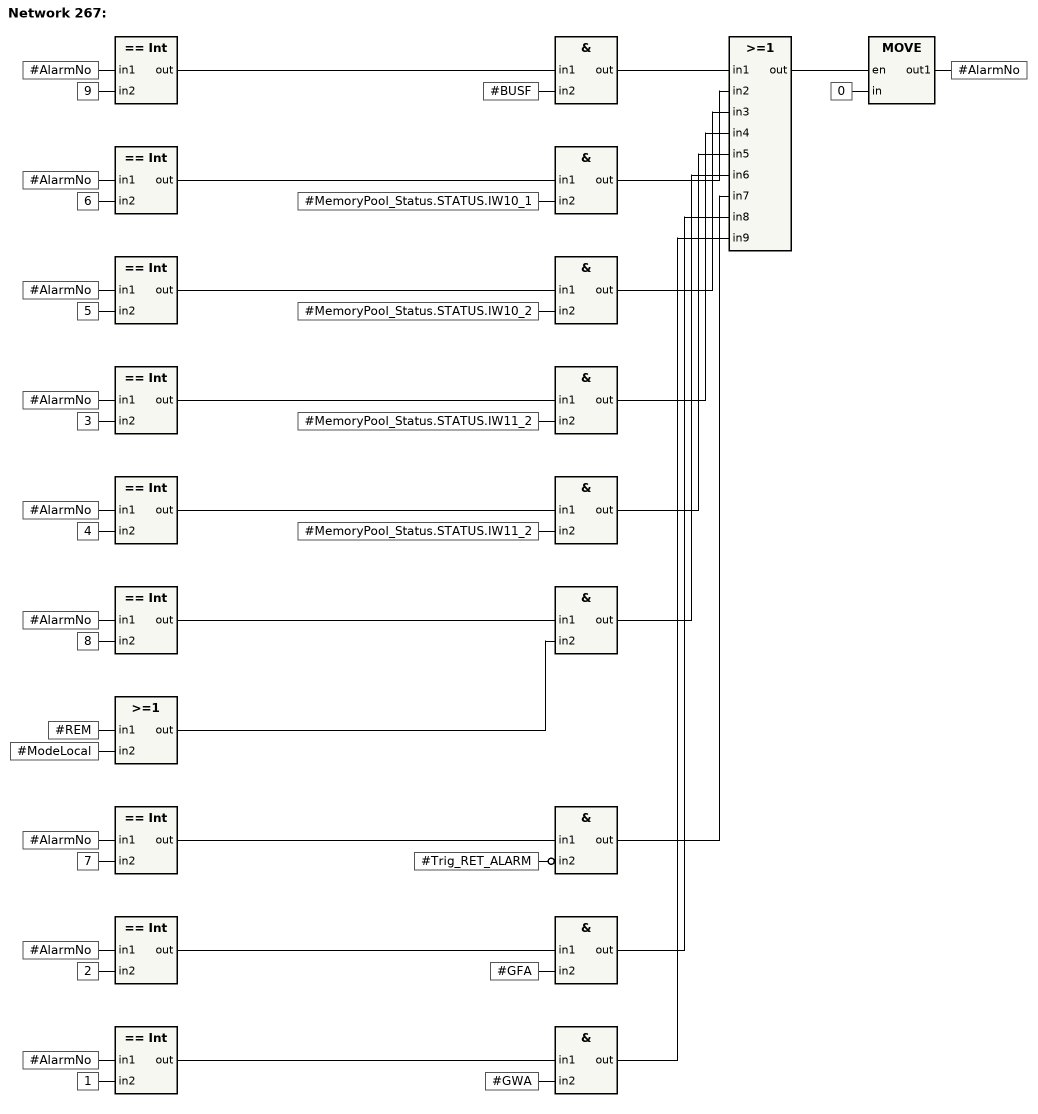
   IF ((#AlarmNo = 9) AND #BUSF) OR ((#AlarmNo = 6) AND #MemoryPool_Status.STATUS.IW10_1) OR ((#AlarmNo = 5) AND #MemoryPool_Status.STATUS.IW10_2) OR ((#AlarmNo = 3) AND #MemoryPool_Status.STATUS.IW11_2) OR ((#AlarmNo = 4) AND #MemoryPool_Status.STATUS.IW11_2) OR ((#AlarmNo = 8) AND (#REM OR #ModeLocal)) OR ((#AlarmNo = 7) AND NOT #Trig_RET_ALARM) OR ((#AlarmNo = 2) AND #GFA) OR ((#AlarmNo = 1) AND #GWA) THEN
       #AlarmNo := 0;
   END_IF;
END_REGION

REGION Network 268
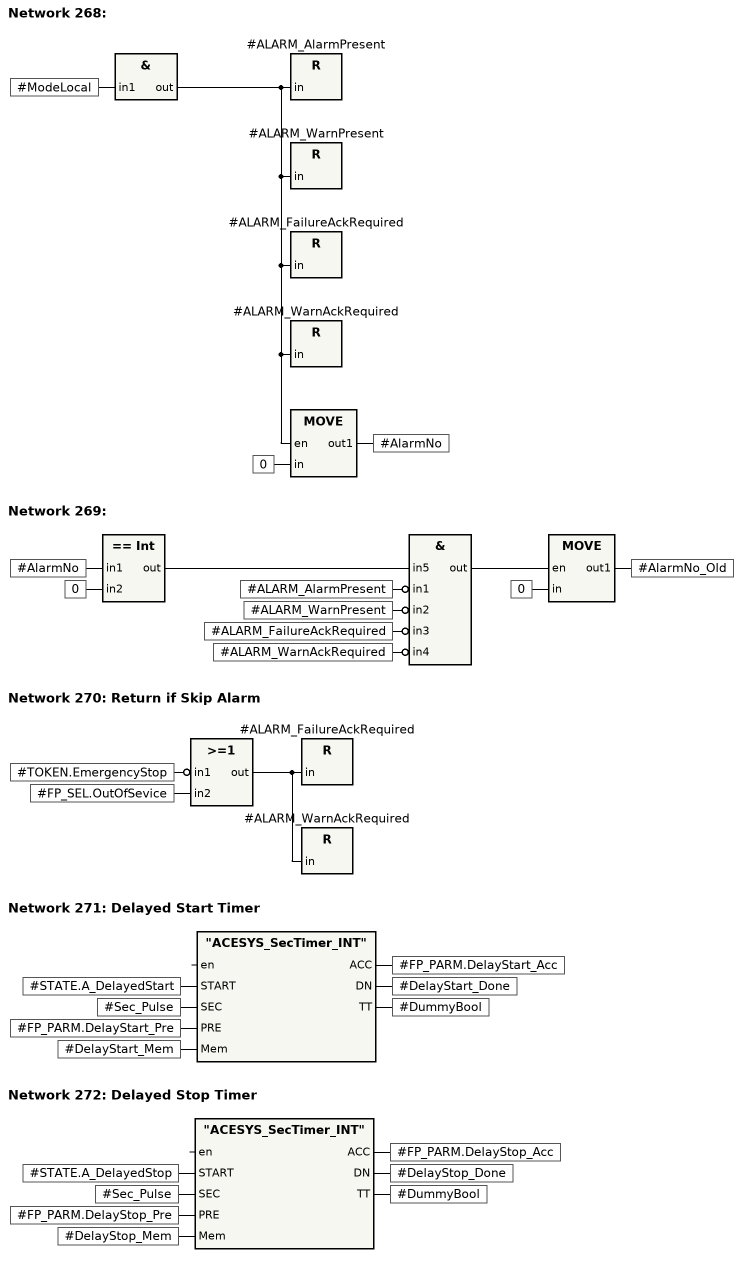
   IF #ModeLocal THEN
       #ALARM_AlarmPresent := FALSE;
       #ALARM_WarnPresent := FALSE;
       #ALARM_FailureAckRequired := FALSE;
       #ALARM_WarnAckRequired := FALSE;
       #AlarmNo := 0;
   END_IF;
END_REGION

REGION Network 269
   IF (#AlarmNo = 0) AND NOT #ALARM_AlarmPresent AND NOT #ALARM_WarnPresent AND NOT #ALARM_FailureAckRequired AND NOT #ALARM_WarnAckRequired THEN
       #AlarmNo_Old := 0;
   END_IF;
END_REGION

REGION Network 270: Return if Skip Alarm
   // Build 002 - 27 March 2019 : Alarm/Warning are Auto Ack on OutOfService
   Skip:
   IF NOT #TOKEN.EmergencyStop OR #FP_SEL.OutOfSevice THEN
       #ALARM_FailureAckRequired := FALSE;
       #ALARM_WarnAckRequired := FALSE;
   END_IF;
END_REGION

REGION Network 271: Delayed Start Timer
   "ACESYS_SecTimer_INT"(START := #STATE.A_DelayedStart,
                         SEC := #Sec_Pulse,
                         PRE := #FP_PARM.DelayStart_Pre,
                         Mem := #DelayStart_Mem,
                         ACC => #FP_PARM.DelayStart_Acc,
                         DN => #DelayStart_Done,
                         TT => #DummyBool);
END_REGION

REGION Network 272: Delayed Stop Timer
   "ACESYS_SecTimer_INT"(START := #STATE.A_DelayedStop,
                         SEC := #Sec_Pulse,
                         PRE := #FP_PARM.DelayStop_Pre,
                         Mem := #DelayStop_Mem,
                         ACC => #FP_PARM.DelayStop_Acc,
                         DN => #DelayStop_Done,
                         TT => #DummyBool);
END_REGION

REGION Network 273: Start Warning timer
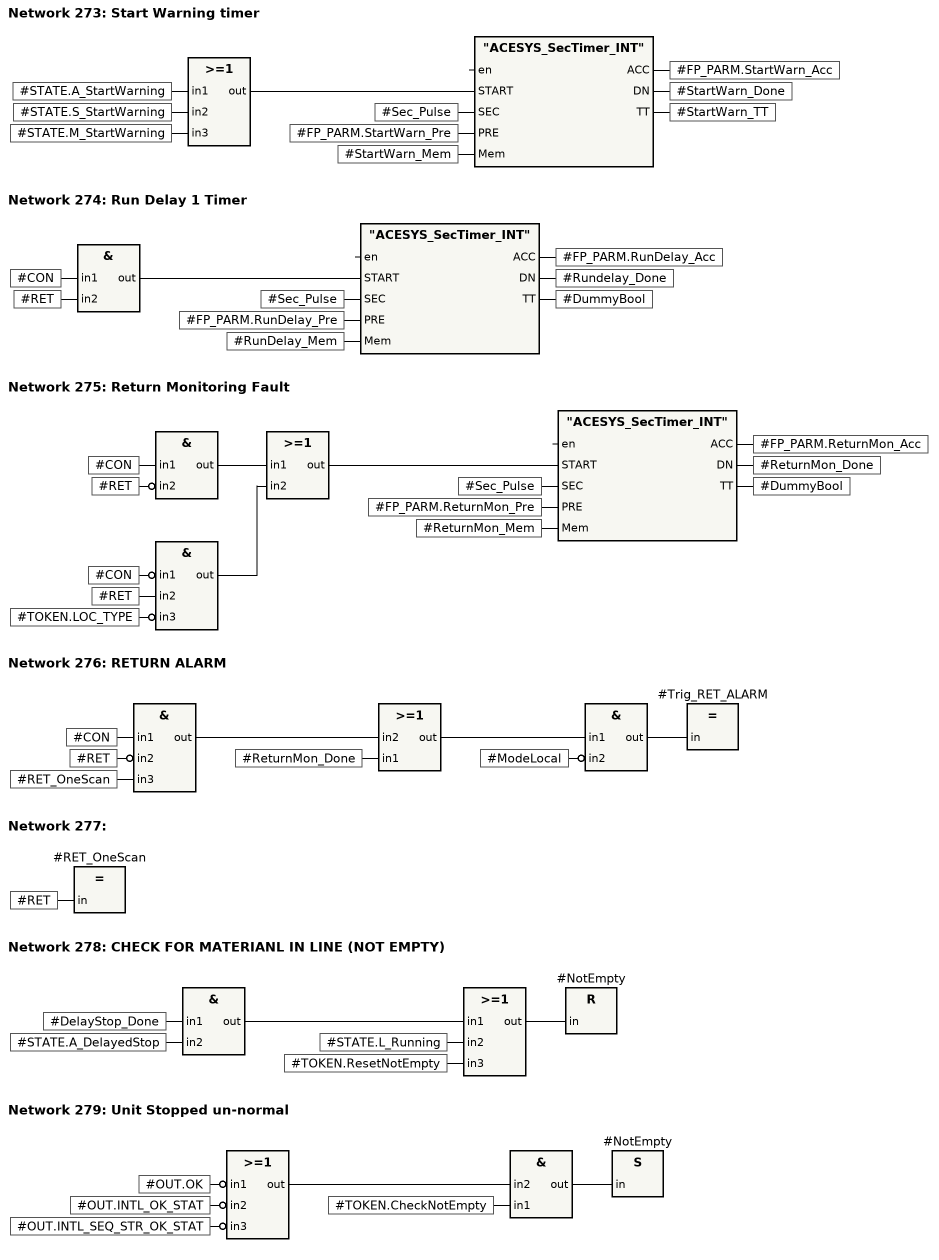
   "ACESYS_SecTimer_INT"(START := #STATE.A_StartWarning OR #STATE.S_StartWarning OR #STATE.M_StartWarning,
                         SEC := #Sec_Pulse,
                         PRE := #FP_PARM.StartWarn_Pre,
                         Mem := #StartWarn_Mem,
                         ACC => #FP_PARM.StartWarn_Acc,
                         DN => #StartWarn_Done,
                         TT => #StartWarn_TT);
END_REGION

REGION Network 274: Run Delay 1 Timer
   "ACESYS_SecTimer_INT"(START := #CON AND #RET,
                         SEC := #Sec_Pulse,
                         PRE := #FP_PARM.RunDelay_Pre,
                         Mem := #RunDelay_Mem,
                         ACC => #FP_PARM.RunDelay_Acc,
                         DN => #Rundelay_Done,
                         TT => #DummyBool);
END_REGION

REGION Network 275: Return Monitoring Fault
   "ACESYS_SecTimer_INT"(START := (#CON AND NOT #RET) OR (NOT #CON AND #RET AND NOT #TOKEN.LOC_TYPE),
                         SEC := #Sec_Pulse,
                         PRE := #FP_PARM.ReturnMon_Pre,
                         Mem := #ReturnMon_Mem,
                         ACC => #FP_PARM.ReturnMon_Acc,
                         DN => #ReturnMon_Done,
                         TT => #DummyBool);
END_REGION

REGION Network 276: RETURN ALARM
   #Trig_RET_ALARM := ((#CON AND NOT #RET AND #RET_OneScan) OR #ReturnMon_Done) AND NOT #ModeLocal;
END_REGION

REGION Network 277
   #RET_OneScan := #RET;
END_REGION

REGION Network 278: CHECK FOR MATERIANL IN LINE (NOT EMPTY)
   IF (#DelayStop_Done AND #STATE.A_DelayedStop) OR #STATE.L_Running OR #TOKEN.ResetNotEmpty THEN
       #NotEmpty := FALSE;
   END_IF;
END_REGION

REGION Network 279: Unit Stopped un-normal
   IF (NOT #OUT.OK OR NOT #OUT.INTL_OK_STAT OR NOT #OUT.INTL_SEQ_STR_OK_STAT) AND #TOKEN.CheckNotEmpty THEN
       #NotEmpty := TRUE;
   END_IF;
END_REGION

REGION Network 280: CHECK FOR STOP REASON & SET OUTPUT COMMANDS
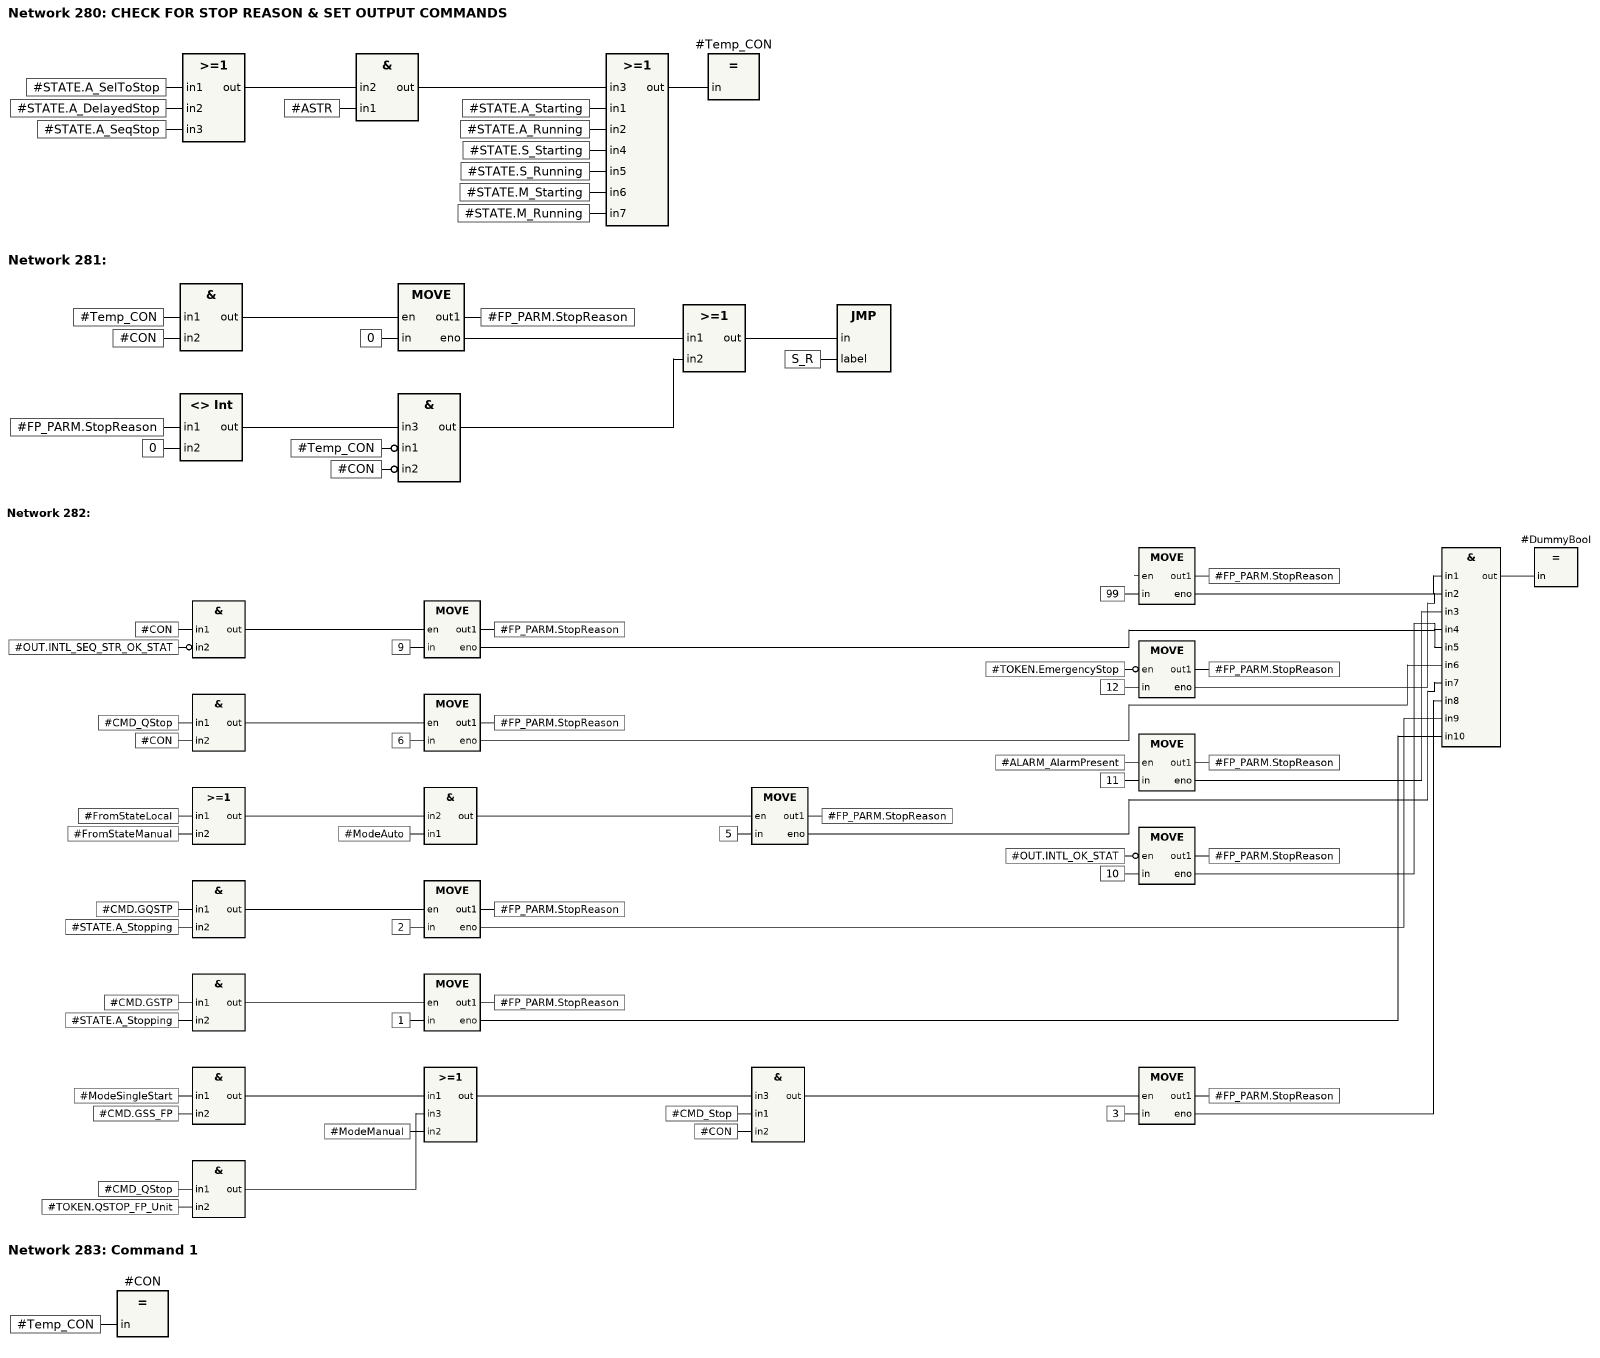
   #Temp_CON := ((#STATE.A_SelToStop OR #STATE.A_DelayedStop OR #STATE.A_SeqStop) AND #ASTR) OR #STATE.A_Starting OR #STATE.A_Running OR #STATE.S_Starting OR #STATE.S_Running OR #STATE.M_Starting OR #STATE.M_Running;
END_REGION

REGION Network 281
   // ENO of a box is taken as its EN; it also drops when the box reports an error
   #_w1 := #Temp_CON AND #CON;
   IF #_w1 THEN #FP_PARM.StopReason := 0; END_IF;
   IF #_w1 OR ((#FP_PARM.StopReason <> 0) AND NOT #Temp_CON AND NOT #CON) THEN GOTO S_R; END_IF;
END_REGION

REGION Network 282
   // 0=In Operation
   // 1=Normal Stop
   // 2=Quick Stop
   // 3=Faceplate Stop
   // 4=Local Stop
   // 5=Change To Auto Mode
   // 6=Quick Stop From Unit Faceplate
   // 9=Sequence Interlock
   // 10=Interlock
   // 11=Unit Alarm
   // 12=Emergency Stop
   // 99=Unknown Reason
   // ENO of a box is taken as its EN; it also drops when the box reports an error
   #FP_PARM.StopReason := 99;
   IF NOT #TOKEN.EmergencyStop THEN #FP_PARM.StopReason := 12; END_IF;
   IF #ALARM_AlarmPresent THEN #FP_PARM.StopReason := 11; END_IF;
   IF NOT #OUT.INTL_OK_STAT THEN #FP_PARM.StopReason := 10; END_IF;
   #_w1 := #CON AND NOT #OUT.INTL_SEQ_STR_OK_STAT;
   IF #_w1 THEN #FP_PARM.StopReason := 9; END_IF;
   #_w2 := #CMD_QStop AND #CON;
   IF #_w2 THEN #FP_PARM.StopReason := 6; END_IF;
   #_w3 := (#FromStateLocal OR #FromStateManual) AND #ModeAuto;
   IF #_w3 THEN #FP_PARM.StopReason := 5; END_IF;
   #_w4 := ((#ModeSingleStart AND #CMD.GSS_FP) OR (#CMD_QStop AND #TOKEN.QSTOP_FP_Unit) OR #ModeManual) AND #CMD_Stop AND #CON;
   IF #_w4 THEN #FP_PARM.StopReason := 3; END_IF;
   #_w5 := #CMD.GQSTP AND #STATE.A_Stopping;
   IF #_w5 THEN #FP_PARM.StopReason := 2; END_IF;
   #_w6 := #CMD.GSTP AND #STATE.A_Stopping;
   IF #_w6 THEN #FP_PARM.StopReason := 1; END_IF;
   #DummyBool := NOT #TOKEN.EmergencyStop AND #ALARM_AlarmPresent AND NOT #OUT.INTL_OK_STAT AND #_w1 AND #_w2 AND #_w3 AND #_w4 AND #_w5 AND #_w6;
END_REGION

REGION Network 283: Command 1
   S_R:
   #CON := #Temp_CON;
END_REGION

REGION Network 284: OUTPUT
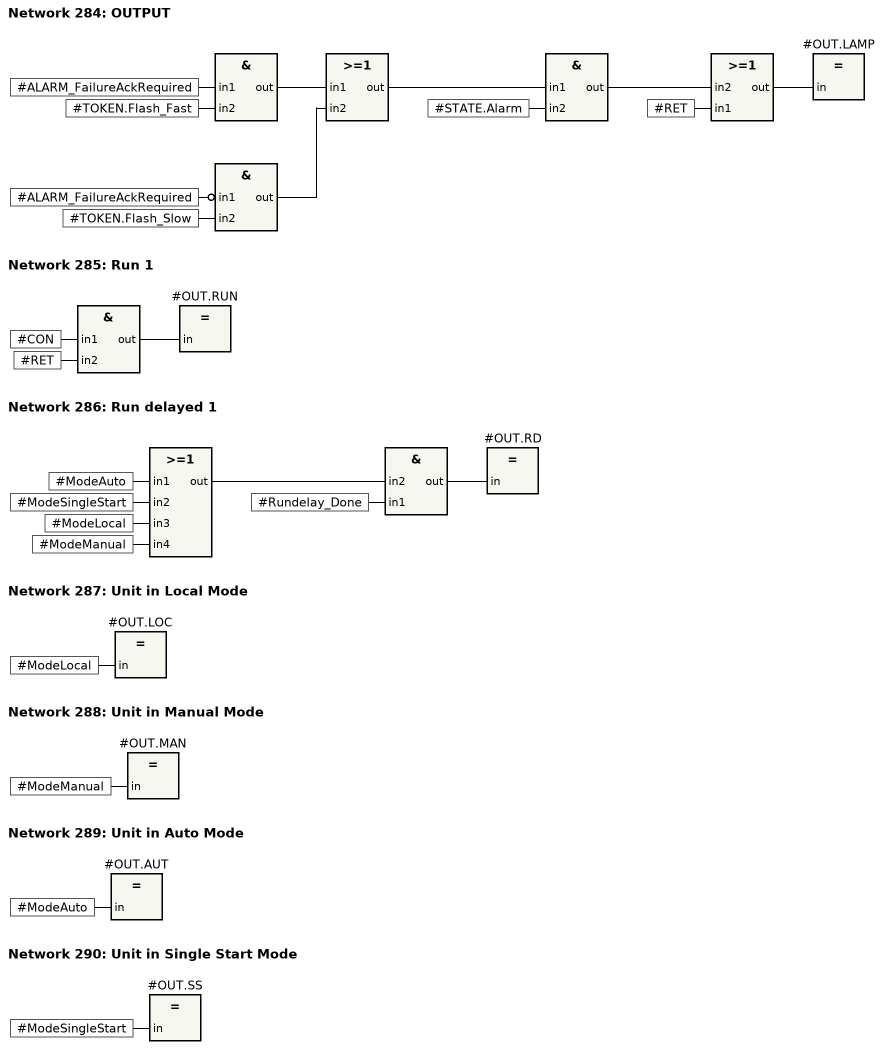
   #OUT.LAMP := (((#ALARM_FailureAckRequired AND #TOKEN.Flash_Fast) OR (NOT #ALARM_FailureAckRequired AND #TOKEN.Flash_Slow)) AND #STATE.Alarm) OR #RET;
END_REGION

REGION Network 285: Run 1
   #OUT.RUN := #CON AND #RET;
END_REGION

REGION Network 286: Run delayed 1
   #OUT.RD := (#ModeAuto OR #ModeSingleStart OR #ModeLocal OR #ModeManual) AND #Rundelay_Done;
END_REGION

REGION Network 287: Unit in Local Mode
   #OUT.LOC := #ModeLocal;
END_REGION

REGION Network 288: Unit in Manual Mode
   #OUT.MAN := #ModeManual;
END_REGION

REGION Network 289: Unit in Auto Mode
   #OUT.AUT := #ModeAuto;
END_REGION

REGION Network 290: Unit in Single Start Mode
   #OUT.SS := #ModeSingleStart;
END_REGION

REGION Network 291: Start Acknowledge
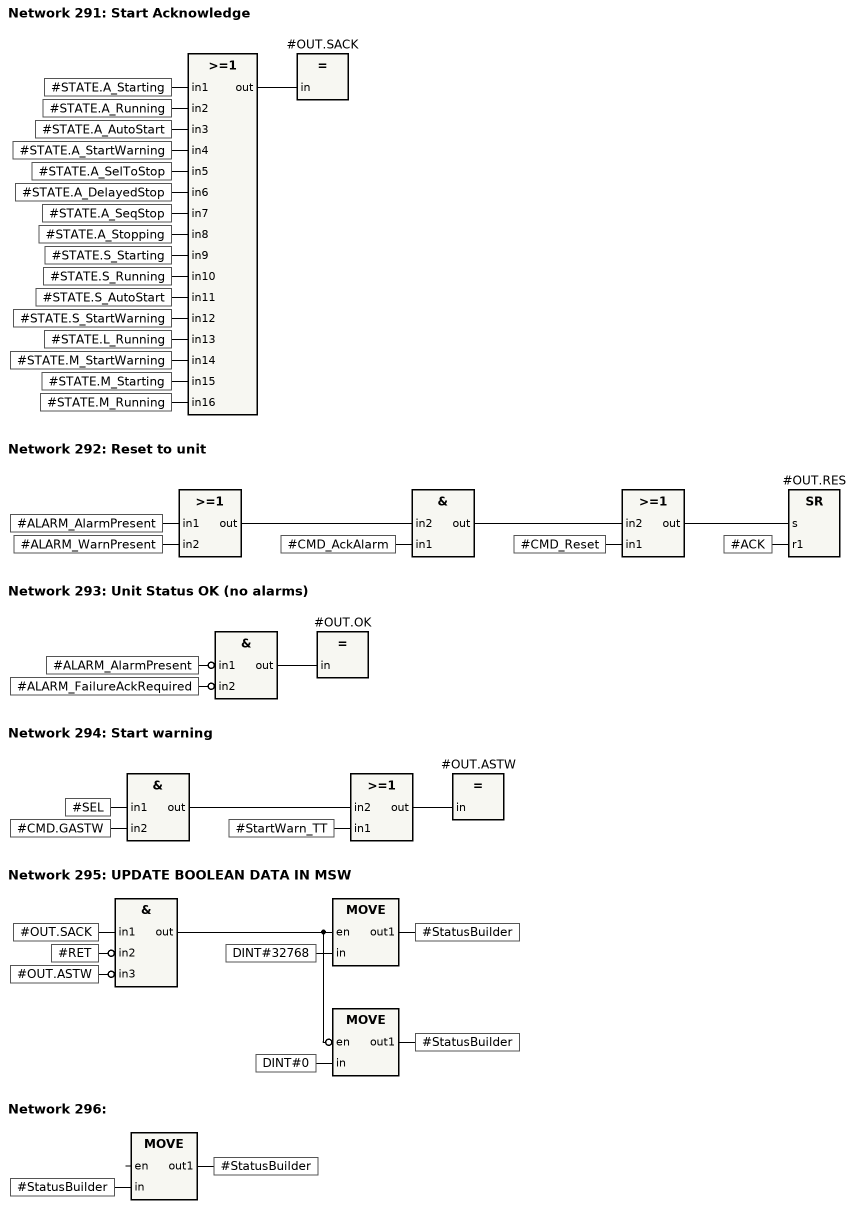
   #OUT.SACK := #STATE.A_Starting OR #STATE.A_Running OR #STATE.A_AutoStart OR #STATE.A_StartWarning OR #STATE.A_SelToStop OR #STATE.A_DelayedStop OR #STATE.A_SeqStop OR #STATE.A_Stopping OR #STATE.S_Starting OR #STATE.S_Running OR #STATE.S_AutoStart OR #STATE.S_StartWarning OR #STATE.L_Running OR #STATE.M_StartWarning OR #STATE.M_Starting OR #STATE.M_Running;
END_REGION

REGION Network 292: Reset to unit
   IF ((#ALARM_AlarmPresent OR #ALARM_WarnPresent) AND #CMD_AckAlarm) OR #CMD_Reset THEN
       #OUT.RES := TRUE;   // SR flip-flop
   END_IF;
   IF #ACK THEN #OUT.RES := FALSE; END_IF;
END_REGION

REGION Network 293: Unit Status OK (no alarms)
   #OUT.OK := NOT #ALARM_AlarmPresent AND NOT #ALARM_FailureAckRequired;
END_REGION

REGION Network 294: Start warning
   #OUT.ASTW := (#SEL AND #CMD.GASTW) OR #StartWarn_TT;
END_REGION

REGION Network 295: UPDATE BOOLEAN DATA IN MSW
   #_w1 := #OUT.SACK AND NOT #RET AND NOT #OUT.ASTW;
   IF #_w1 THEN #StatusBuilder := DINT#32768; END_IF;
   IF NOT #_w1 THEN #StatusBuilder := DINT#0; END_IF;
END_REGION

REGION Network 296
   #StatusBuilder := #StatusBuilder;
END_REGION

REGION Network 297: Bit 16: Mode bit 1 (value = 1)
